    //FB-s
    EL3255_Error    : FB_TerminalError;
    CH1_Error       : FB_GenericError;
    CH2_Error       : FB_GenericError;
    CH3_Error       : FB_GenericError;
    CH4_Error       : FB_GenericError;
    CH5_Error       : FB_GenericError;
END_VAR

(*
* TODO: Test on hardware
*)
EnO:=En;

IF En THEN
    //Channel #1 Status
    IF (wCh1_Status AND 16#2057) <> 0 THEN
        CH1_Error.sErrorMessage := 'EL3255 Channel #1: ';
        IF wCH1_Status.0    THEN    CH1_Error.sErrorMessage := CONCAT(CH1_Error.sErrorMessage, 'Underrange; ');             IF CH1_Error.ErrorPriority > 100 OR CH1_Error.ErrorPriority = 0     THEN CH1_Error.ErrorPriority := 100;    END_IF      END_IF
        IF wCH1_Status.1    THEN    CH1_Error.sErrorMessage := CONCAT(CH1_Error.sErrorMessage, 'Overrange; ');              IF CH1_Error.ErrorPriority > 100 OR CH1_Error.ErrorPriority = 0     THEN CH1_Error.ErrorPriority := 100;    END_IF      END_IF
        IF wCh1_Status.2    THEN    CH1_Error.sErrorMessage := CONCAT(CH1_Error.sErrorMessage, 'Limit 1; ');                IF CH1_Error.ErrorPriority > 100 OR CH1_Error.ErrorPriority = 0     THEN CH1_Error.ErrorPriority := 100;    END_IF      END_IF
        IF wCh1_Status.4    THEN    CH1_Error.sErrorMessage := CONCAT(CH1_Error.sErrorMessage, 'Limit 2; ');                IF CH1_Error.ErrorPriority > 100 OR CH1_Error.ErrorPriority = 0     THEN CH1_Error.ErrorPriority := 100;    END_IF      END_IF
        IF wCh1_Status.6    THEN    CH1_Error.sErrorMessage := CONCAT(CH1_Error.sErrorMessage, 'Error; ');                  IF CH1_Error.ErrorPriority > 10  OR CH1_Error.ErrorPriority = 0     THEN CH1_Error.ErrorPriority := 10;     END_IF      END_IF
        IF wCh1_Status.13   THEN    CH1_Error.sErrorMessage := CONCAT(CH1_Error.sErrorMessage, 'Sync error; ');             IF CH1_Error.ErrorPriority > 10  OR CH1_Error.ErrorPriority = 0     THEN CH1_Error.ErrorPriority := 10;     END_IF      END_IF
        CH1_Error.bError := TRUE;
    ELSE
        CH1_Error.bError        := FALSE;
        CH1_Error.sErrorMessage := '';
    END_IF

    //Channel #2 Status
    IF (wCh2_Status AND 16#2057) <> 0 THEN
        CH2_Error.sErrorMessage := 'EL3255 Channel #2: ';
        IF wCH2_Status.0    THEN    CH2_Error.sErrorMessage := CONCAT(CH2_Error.sErrorMessage, 'Underrange; ');             IF CH2_Error.ErrorPriority > 100 OR CH2_Error.ErrorPriority = 0     THEN CH2_Error.ErrorPriority := 100;    END_IF      END_IF
        IF wCH2_Status.1    THEN    CH2_Error.sErrorMessage := CONCAT(CH2_Error.sErrorMessage, 'Overrange; ');              IF CH2_Error.ErrorPriority > 100 OR CH2_Error.ErrorPriority = 0     THEN CH2_Error.ErrorPriority := 100;    END_IF      END_IF
        IF wCh2_Status.2    THEN    CH2_Error.sErrorMessage := CONCAT(CH2_Error.sErrorMessage, 'Limit 1; ');                IF CH2_Error.ErrorPriority > 100 OR CH2_Error.ErrorPriority = 0     THEN CH2_Error.ErrorPriority := 100;    END_IF      END_IF
        IF wCh2_Status.4    THEN    CH2_Error.sErrorMessage := CONCAT(CH2_Error.sErrorMessage, 'Limit 2; ');                IF CH2_Error.ErrorPriority > 100 OR CH2_Error.ErrorPriority = 0     THEN CH2_Error.ErrorPriority := 100;    END_IF      END_IF
        IF wCh2_Status.6    THEN    CH2_Error.sErrorMessage := CONCAT(CH2_Error.sErrorMessage, 'Error; ');                  IF CH2_Error.ErrorPriority > 10  OR CH2_Error.ErrorPriority = 0     THEN CH2_Error.ErrorPriority := 10;     END_IF      END_IF
        IF wCh2_Status.13   THEN    CH2_Error.sErrorMessage := CONCAT(CH2_Error.sErrorMessage, 'Sync error; ');             IF CH2_Error.ErrorPriority > 10  OR CH2_Error.ErrorPriority = 0     THEN CH2_Error.ErrorPriority := 10;     END_IF      END_IF
        CH2_Error.bError := TRUE;
    ELSE
        CH2_Error.bError        := FALSE;
        CH2_Error.sErrorMessage := '';
    END_IF

    //Channel #3 Status
    IF (wCh3_Status AND 16#2057) <> 0 THEN
        CH3_Error.sErrorMessage := 'EL3255 Channel #3: ';
        IF wCH3_Status.0    THEN    CH3_Error.sErrorMessage := CONCAT(CH3_Error.sErrorMessage, 'Underrange; ');             IF CH3_Error.ErrorPriority > 100 OR CH3_Error.ErrorPriority = 0     THEN CH3_Error.ErrorPriority := 100;    END_IF      END_IF
        IF wCH3_Status.1    THEN    CH3_Error.sErrorMessage := CONCAT(CH3_Error.sErrorMessage, 'Overrange; ');              IF CH3_Error.ErrorPriority > 100 OR CH3_Error.ErrorPriority = 0     THEN CH3_Error.ErrorPriority := 100;    END_IF      END_IF
        IF wCh3_Status.2    THEN    CH3_Error.sErrorMessage := CONCAT(CH3_Error.sErrorMessage, 'Limit 1; ');                IF CH3_Error.ErrorPriority > 100 OR CH3_Error.ErrorPriority = 0     THEN CH3_Error.ErrorPriority := 100;    END_IF      END_IF
        IF wCh3_Status.4    THEN    CH3_Error.sErrorMessage := CONCAT(CH3_Error.sErrorMessage, 'Limit 2; ');                IF CH3_Error.ErrorPriority > 100 OR CH3_Error.ErrorPriority = 0     THEN CH3_Error.ErrorPriority := 100;    END_IF      END_IF
        IF wCh3_Status.6    THEN    CH3_Error.sErrorMessage := CONCAT(CH3_Error.sErrorMessage, 'Error; ');                  IF CH3_Error.ErrorPriority > 10  OR CH3_Error.ErrorPriority = 0     THEN CH3_Error.ErrorPriority := 10;     END_IF      END_IF
        IF wCh3_Status.13   THEN    CH3_Error.sErrorMessage := CONCAT(CH3_Error.sErrorMessage, 'Sync error; ');             IF CH3_Error.ErrorPriority > 10  OR CH3_Error.ErrorPriority = 0     THEN CH3_Error.ErrorPriority := 10;     END_IF      END_IF
        CH3_Error.bError := TRUE;
    ELSE
        CH3_Error.bError        := FALSE;
        CH3_Error.sErrorMessage := '';
    END_IF

    //Channel #4 Status
    IF (wCh4_Status AND 16#2057) <> 0 THEN
        CH4_Error.sErrorMessage := 'EL3255 Channel #4: ';
        IF wCH4_Status.0    THEN    CH4_Error.sErrorMessage := CONCAT(CH4_Error.sErrorMessage, 'Underrange; ');             IF CH4_Error.ErrorPriority > 100 OR CH4_Error.ErrorPriority = 0     THEN CH4_Error.ErrorPriority := 100;    END_IF      END_IF
        IF wCH4_Status.1    THEN    CH4_Error.sErrorMessage := CONCAT(CH4_Error.sErrorMessage, 'Overrange; ');              IF CH4_Error.ErrorPriority > 100 OR CH4_Error.ErrorPriority = 0     THEN CH4_Error.ErrorPriority := 100;    END_IF      END_IF
        IF wCh4_Status.2    THEN    CH4_Error.sErrorMessage := CONCAT(CH4_Error.sErrorMessage, 'Limit 1; ');                IF CH4_Error.ErrorPriority > 100 OR CH4_Error.ErrorPriority = 0     THEN CH4_Error.ErrorPriority := 100;    END_IF      END_IF
        IF wCh4_Status.4    THEN    CH4_Error.sErrorMessage := CONCAT(CH4_Error.sErrorMessage, 'Limit 2; ');                IF CH4_Error.ErrorPriority > 100 OR CH4_Error.ErrorPriority = 0     THEN CH4_Error.ErrorPriority := 100;    END_IF      END_IF
        IF wCh4_Status.6    THEN    CH4_Error.sErrorMessage := CONCAT(CH4_Error.sErrorMessage, 'Error; ');                  IF CH4_Error.ErrorPriority > 10  OR CH4_Error.ErrorPriority = 0     THEN CH4_Error.ErrorPriority := 10;     END_IF      END_IF
        IF wCh4_Status.13   THEN    CH4_Error.sErrorMessage := CONCAT(CH4_Error.sErrorMessage, 'Sync error; ');             IF CH4_Error.ErrorPriority > 10  OR CH4_Error.ErrorPriority = 0     THEN CH4_Error.ErrorPriority := 10;     END_IF      END_IF
        CH4_Error.bError := TRUE;
    ELSE
        CH4_Error.bError        := FALSE;
        CH4_Error.sErrorMessage := '';
    END_IF

    //Channel #5 Status
    IF (wCh5_Status AND 16#2057) <> 0 THEN
        CH5_Error.sErrorMessage := 'EL3255 Channel #5: ';
        IF wCH5_Status.0    THEN    CH5_Error.sErrorMessage := CONCAT(CH5_Error.sErrorMessage, 'Underrange; ');             IF CH5_Error.ErrorPriority > 100 OR CH5_Error.ErrorPriority = 0     THEN CH5_Error.ErrorPriority := 100;    END_IF      END_IF
        IF wCH5_Status.1    THEN    CH5_Error.sErrorMessage := CONCAT(CH5_Error.sErrorMessage, 'Overrange; ');              IF CH5_Error.ErrorPriority > 100 OR CH5_Error.ErrorPriority = 0     THEN CH5_Error.ErrorPriority := 100;    END_IF      END_IF
        IF wCh5_Status.2    THEN    CH5_Error.sErrorMessage := CONCAT(CH5_Error.sErrorMessage, 'Limit 1; ');                IF CH5_Error.ErrorPriority > 100 OR CH5_Error.ErrorPriority = 0     THEN CH5_Error.ErrorPriority := 100;    END_IF      END_IF
        IF wCh5_Status.4    THEN    CH5_Error.sErrorMessage := CONCAT(CH5_Error.sErrorMessage, 'Limit 2; ');                IF CH5_Error.ErrorPriority > 100 OR CH5_Error.ErrorPriority = 0     THEN CH5_Error.ErrorPriority := 100;    END_IF      END_IF
        IF wCh5_Status.6    THEN    CH5_Error.sErrorMessage := CONCAT(CH5_Error.sErrorMessage, 'Error; ');                  IF CH5_Error.ErrorPriority > 10  OR CH5_Error.ErrorPriority = 0     THEN CH5_Error.ErrorPriority := 10;     END_IF      END_IF
        IF wCh5_Status.13   THEN    CH5_Error.sErrorMessage := CONCAT(CH5_Error.sErrorMessage, 'Sync error; ');             IF CH5_Error.ErrorPriority > 10  OR CH5_Error.ErrorPriority = 0     THEN CH5_Error.ErrorPriority := 10;     END_IF      END_IF
        CH5_Error.bError := TRUE;
    ELSE
        CH5_Error.bError        := FALSE;
        CH5_Error.sErrorMessage := '';
    END_IF

END_IF

//Error FB instance
EL3255_Error(
    En                  := TRUE,
    iTerminal_ID        := iTerminal_ID,
    bWcState            := WcState_WcState,
    uiInfoData_State    := InfoData_State,
    pErrorSystem        := ErrorSystem,
    bError              => bError,
);

CH1_Error (
    En              := En,
    bError          := ,
    sErrorMessage   := ,
    ErrorPriority   := ,
    iTerminal_ID    := iTerminal_ID,
    pErrorSystem    := ErrorSystem,
    EnO             => ,
);

CH2_Error (
    En              := En,
    bError          := ,
    sErrorMessage   := ,
    ErrorPriority   := ,
    iTerminal_ID    := iTerminal_ID,
    pErrorSystem    := ErrorSystem,
    EnO             => ,
);

CH3_Error (
    En              := En,
    bError          := ,
    sErrorMessage   := ,
    ErrorPriority   := ,
    iTerminal_ID    := iTerminal_ID,
    pErrorSystem    := ErrorSystem,
    EnO             => ,
);

CH4_Error (
    En              := En,
    bError          := ,
    sErrorMessage   := ,
    ErrorPriority   := ,
    iTerminal_ID    := iTerminal_ID,
    pErrorSystem    := ErrorSystem,
    EnO             => ,
);

CH5_Error (
    En              := En,
    bError          := ,
    sErrorMessage   := ,
    ErrorPriority   := ,
    iTerminal_ID    := iTerminal_ID,
    pErrorSystem    := ErrorSystem,
    EnO             => ,
);

END_FUNCTION_BLOCK

// ---- tc_mca_std_lib/POUs/Hardware/EtherCAT_Terminals/Digital_Inputs/EL1008.TcPOU
///EL1008 | 8-channel digital input terminal 24 V DC, 3 ms
FUNCTION_BLOCK EL1008

VAR_INPUT
    En              : BOOL;
    iTerminal_ID    : INT;
    ErrorSystem     : POINTER TO ST_ErrorSystem;
END_VAR

VAR_OUTPUT
    EnO     : BOOL;
    bError  : BOOL;
END_VAR

VAR
    WcState_WcState     AT %I*  : BOOL;
    InfoData_State      AT %I*  : UINT;

    //FB-s
    EL1008_Error    : FB_TerminalError;
END_VAR

(*
* TODO: DONE!
*)
EnO:=En;

//Error FB instance
EL1008_Error(
    En                  := TRUE,
    iTerminal_ID        := iTerminal_ID,
    bWcState            := WcState_WcState,
    uiInfoData_State    := InfoData_State,
    pErrorSystem        := ErrorSystem,
    bError              => bError,
);

END_FUNCTION_BLOCK

// ---- tc_mca_std_lib/POUs/Hardware/EtherCAT_Terminals/Digital_Inputs/EL1018.TcPOU
///EL1018 | 8-channel digital input terminal 24 V DC, 10 µs
FUNCTION_BLOCK EL1018

VAR_INPUT
    En              : BOOL;
    iTerminal_ID    : INT;
    ErrorSystem     : POINTER TO ST_ErrorSystem;
END_VAR

VAR_OUTPUT
    EnO         : BOOL;
    bError      : BOOL;
END_VAR

VAR
    WcState_WcState     AT %I*  : BOOL;
    InfoData_State      AT %I*  : UINT;

    //FB-s
    EL1018_Error    : FB_TerminalError;
END_VAR

(*
* TODO: DONE!
*)
EnO:=En;

//Error FB instance
EL1018_Error(
    En                  := TRUE,
    iTerminal_ID        := iTerminal_ID,
    bWcState            := WcState_WcState,
    uiInfoData_State    := InfoData_State,
    pErrorSystem        := ErrorSystem,
    bError              => bError,
);

END_FUNCTION_BLOCK

// ---- tc_mca_std_lib/POUs/Hardware/EtherCAT_Terminals/Digital_Inputs/EL1252.TcPOU
//EL1252 or EL1252-0050 | 2-channel digitl input terminal with timestamp
FUNCTION_BLOCK EL1252
VAR_INPUT
    En              : BOOL;
    iTerminal_ID    : INT;
    ErrorSystem     : POINTER TO ST_ErrorSystem;
END_VAR

VAR_OUTPUT
    EnO     : BOOL;
    bError  : BOOL;
END_VAR

VAR
    WcState_WcState     AT %I*  : BOOL;
    InfoData_State      AT %I*  : UINT;

    //FB-s
    EL1252_Error        : FB_TerminalError;
END_VAR

(*
* TODO: DONE!
*)
EnO:=En;

//Error FB instance
EL1252_Error(
    En                  := TRUE,
    iTerminal_ID        := iTerminal_ID,
    bWcState            := WcState_WcState,
    uiInfoData_State    := InfoData_State,
    pErrorSystem        := ErrorSystem,
    bError              => bError,
);

END_FUNCTION_BLOCK

// ---- tc_mca_std_lib/POUs/Hardware/EtherCAT_Terminals/Digital_Inputs/EL1808.TcPOU
///EL1808 | HD EtherCAT Terminals, 8-channel digital input 24 V DC, 3 ms, 2-wire connection
FUNCTION_BLOCK EL1808

VAR_INPUT
    En              : BOOL;
    iTerminal_ID    : INT;
    ErrorSystem     : POINTER TO ST_ErrorSystem;
END_VAR

VAR_OUTPUT
    EnO         : BOOL;
    bError      : BOOL;
END_VAR

VAR
    WcState_WcState     AT %I*  : BOOL;
    InfoData_State      AT %I*  : UINT;

    //FB-s
    EL1808_Error    : FB_TerminalError;
END_VAR

(*
* TODO: DONE!
*)
EnO:=En;

//Error FB instance
EL1808_Error(
    En                  := TRUE,
    iTerminal_ID        := iTerminal_ID,
    bWcState            := WcState_WcState,
    uiInfoData_State    := InfoData_State,
    pErrorSystem        := ErrorSystem,
    bError              => bError,
);

END_FUNCTION_BLOCK

// ---- tc_mca_std_lib/POUs/Hardware/EtherCAT_Terminals/Digital_Inputs/EL1809.TcPOU
///EL1809 | HD EtherCAT Terminals, 16-channel digital input 24 V DC, 3 ms
FUNCTION_BLOCK EL1809

VAR_INPUT
    En              : BOOL;
    iTerminal_ID    : INT;
    ErrorSystem     : POINTER TO ST_ErrorSystem;
END_VAR

VAR_OUTPUT
    EnO     : BOOL;
    bError  : BOOL;
END_VAR

VAR
    WcState_WcState     AT %I*  : BOOL;
    InfoData_State      AT %I*  : UINT;

    //FB-s
    EL1809_Error    : FB_TerminalError;
END_VAR

(*
* TODO: DONE!
*)
EnO:=En;

//Error FB instance
EL1809_Error(
    En                  := TRUE,
    iTerminal_ID        := iTerminal_ID,
    bWcState            := WcState_WcState,
    uiInfoData_State    := InfoData_State,
    pErrorSystem        := ErrorSystem,
    bError              => bError,
);

END_FUNCTION_BLOCK

// ---- tc_mca_std_lib/POUs/Hardware/EtherCAT_Terminals/Digital_Inputs/EL1819.TcPOU
///EL1819 | HD EtherCAT Terminals, 16-channel digital input 24 V DC, 10 µs
FUNCTION_BLOCK EL1819

VAR_INPUT
    En              : BOOL;
    iTerminal_ID    : INT;
    ErrorSystem     : POINTER TO ST_ErrorSystem;
END_VAR

VAR_OUTPUT
    EnO         : BOOL;
    bError      : BOOL;
END_VAR

VAR
    WcState_WcState     AT %I*  : BOOL;
    InfoData_State      AT %I*  : UINT;

    //FB-s
    EL1819_Error    : FB_TerminalError;
END_VAR

(*
* TODO: DONE!
*)
EnO:=En;

//Error FB instance
EL1819_Error(
    En                  := TRUE,
    iTerminal_ID        := iTerminal_ID,
    bWcState            := WcState_WcState,
    uiInfoData_State    := InfoData_State,
    pErrorSystem        := ErrorSystem,
    bError              => bError,
);

END_FUNCTION_BLOCK

// ---- tc_mca_std_lib/POUs/Hardware/EtherCAT_Terminals/Digital_Outputs/EL2014.TcPOU
// EL2014 | 4-channel output terminal, 24V DC, 0.5A, 4 x 0V contact
FUNCTION_BLOCK EL2014
VAR_INPUT
    En              : BOOL;
    iTerminal_ID    : INT;
    ErrorSystem     : POINTER TO ST_ErrorSystem;
END_VAR

VAR_OUTPUT
    EnO         : BOOL;
    bError      : BOOL;
END_VAR

VAR
    //Channel Diagnostic Inputs
    wCH1_Diag       AT %I*  : BYTE;
    wCH2_Diag       AT %I*  : BYTE;
    wCH3_Diag       AT %I*  : BYTE;
    wCH4_Diag       AT %I*  : BYTE;
    //Device Diagnostic Inputs
    wDevice_Diag        AT %I*  : BYTE;
    //Device State Inputs
    WcState_WcState     AT %I*  : BOOL;
    InfoData_State      AT %I*  : UINT;


    //FB-s
    EL2014_Error    : FB_TerminalError;
    CH1_Error       : FB_GenericError;
    CH2_Error       : FB_GenericError;
    CH3_Error       : FB_GenericError;
    CH4_Error       : FB_GenericError;
    DEV_Error       : FB_GenericError;
END_VAR

(*
*   TODO: Test on hardware
*)
EnO:=En;

IF En THEN

    //Channel #1 Diag
    IF wCH1_Diag <> 0 THEN
        CH1_Error.sErrorMessage := 'EL2014 Channel #1: ';
        IF wCH1_Diag.0  THEN    CH1_Error.sErrorMessage := CONCAT(CH1_Error.sErrorMessage, 'Overtemperature; ');            IF CH1_Error.ErrorPriority > 10  OR CH1_Error.ErrorPriority = 0     THEN CH1_Error.ErrorPriority := 10;     END_IF      END_IF
        IF wCH1_Diag.1  THEN    CH1_Error.sErrorMessage := CONCAT(CH1_Error.sErrorMessage, 'Open Load; ');                  IF CH1_Error.ErrorPriority > 100 OR CH1_Error.ErrorPriority = 0     THEN CH1_Error.ErrorPriority := 100;    END_IF      END_IF
        IF wCH1_Diag.2  THEN    CH1_Error.sErrorMessage := CONCAT(CH1_Error.sErrorMessage, 'Overcurrent; ');                IF CH1_Error.ErrorPriority > 10  OR CH1_Error.ErrorPriority = 0     THEN CH1_Error.ErrorPriority := 10;     END_IF      END_IF
        IF wCH1_Diag.3  THEN    CH1_Error.sErrorMessage := CONCAT(CH1_Error.sErrorMessage, 'Short Circuit to 24V; ');       IF CH1_Error.ErrorPriority > 10  OR CH1_Error.ErrorPriority = 0     THEN CH1_Error.ErrorPriority := 10;     END_IF      END_IF
        CH1_Error.bError := TRUE;
    ELSE
        CH1_Error.bError := FALSE;
        CH1_Error.sErrorMessage := '';
    END_IF

    //Channel #2 Diag
    IF wCH2_Diag <> 0 THEN
        CH2_Error.sErrorMessage := 'EL2014 Channel #2: ';
        IF wCH2_Diag.0  THEN    CH2_Error.sErrorMessage := CONCAT(CH2_Error.sErrorMessage, 'Overtemperature; ');            IF CH2_Error.ErrorPriority > 10  OR CH2_Error.ErrorPriority = 0     THEN CH2_Error.ErrorPriority := 10;     END_IF      END_IF
        IF wCH2_Diag.1  THEN    CH2_Error.sErrorMessage := CONCAT(CH2_Error.sErrorMessage, 'Open Load; ');                  IF CH2_Error.ErrorPriority > 100 OR CH2_Error.ErrorPriority = 0     THEN CH2_Error.ErrorPriority := 100;    END_IF      END_IF
        IF wCH2_Diag.2  THEN    CH2_Error.sErrorMessage := CONCAT(CH2_Error.sErrorMessage, 'Overcurrent; ');                IF CH2_Error.ErrorPriority > 10  OR CH2_Error.ErrorPriority = 0     THEN CH2_Error.ErrorPriority := 10;     END_IF      END_IF
        IF wCH2_Diag.3  THEN    CH2_Error.sErrorMessage := CONCAT(CH2_Error.sErrorMessage, 'Short Circuit to 24V; ');       IF CH2_Error.ErrorPriority > 10  OR CH2_Error.ErrorPriority = 0     THEN CH2_Error.ErrorPriority := 10;     END_IF      END_IF
        CH2_Error.bError := TRUE;
    ELSE
        CH2_Error.bError := FALSE;
        CH2_Error.sErrorMessage := '';
    END_IF

    //Channel #3 Diag
    IF wCH3_Diag <> 0 THEN
        CH3_Error.sErrorMessage := 'EL2014 Channel #3: ';
        IF wCH3_Diag.0  THEN    CH3_Error.sErrorMessage := CONCAT(CH3_Error.sErrorMessage, 'Overtemperature; ');            IF CH3_Error.ErrorPriority > 10  OR CH3_Error.ErrorPriority = 0     THEN CH3_Error.ErrorPriority := 10;     END_IF      END_IF
        IF wCH3_Diag.1  THEN    CH3_Error.sErrorMessage := CONCAT(CH3_Error.sErrorMessage, 'Open Load; ');                  IF CH3_Error.ErrorPriority > 100 OR CH3_Error.ErrorPriority = 0     THEN CH3_Error.ErrorPriority := 100;    END_IF      END_IF
        IF wCH3_Diag.2  THEN    CH3_Error.sErrorMessage := CONCAT(CH3_Error.sErrorMessage, 'Overcurrent; ');                IF CH3_Error.ErrorPriority > 10  OR CH3_Error.ErrorPriority = 0     THEN CH3_Error.ErrorPriority := 10;     END_IF      END_IF
        IF wCH3_Diag.3  THEN    CH3_Error.sErrorMessage := CONCAT(CH3_Error.sErrorMessage, 'Short Circuit to 24V; ');       IF CH3_Error.ErrorPriority > 10  OR CH3_Error.ErrorPriority = 0     THEN CH3_Error.ErrorPriority := 10;     END_IF      END_IF
        CH3_Error.bError := TRUE;
    ELSE
        CH3_Error.bError := FALSE;
        CH3_Error.sErrorMessage := '';
    END_IF

    //Channel #4 Diag
    IF wCH4_Diag <> 0 THEN
        CH4_Error.sErrorMessage := 'EL2014 Channel #4: ';
        IF wCH4_Diag.0  THEN    CH4_Error.sErrorMessage := CONCAT(CH4_Error.sErrorMessage, 'Overtemperature; ');            IF CH4_Error.ErrorPriority > 10  OR CH4_Error.ErrorPriority = 0     THEN CH4_Error.ErrorPriority := 10;     END_IF      END_IF
        IF wCH4_Diag.1  THEN    CH4_Error.sErrorMessage := CONCAT(CH4_Error.sErrorMessage, 'Open Load; ');                  IF CH4_Error.ErrorPriority > 100 OR CH4_Error.ErrorPriority = 0     THEN CH4_Error.ErrorPriority := 100;    END_IF      END_IF
        IF wCH4_Diag.2  THEN    CH4_Error.sErrorMessage := CONCAT(CH4_Error.sErrorMessage, 'Overcurrent; ');                IF CH4_Error.ErrorPriority > 10  OR CH4_Error.ErrorPriority = 0     THEN CH4_Error.ErrorPriority := 10;     END_IF      END_IF
        IF wCH4_Diag.3  THEN    CH4_Error.sErrorMessage := CONCAT(CH4_Error.sErrorMessage, 'Short Circuit to 24V; ');       IF CH4_Error.ErrorPriority > 10  OR CH4_Error.ErrorPriority = 0     THEN CH4_Error.ErrorPriority := 10;     END_IF      END_IF
        CH4_Error.bError := TRUE;
    ELSE
        CH4_Error.bError := FALSE;
        CH4_Error.sErrorMessage := '';
    END_IF

    //Device Diag
    IF wDevice_Diag <> 0 THEN
        DEV_Error.sErrorMessage := 'EL2014: ' ;
        IF wDevice_Diag.0   THEN    DEV_Error.sErrorMessage := CONCAT(DEV_Error.sErrorMessage, 'Common Fault; ');                   IF DEV_Error.ErrorPriority > 100 OR DEV_Error.ErrorPriority = 0     THEN DEV_Error.ErrorPriority := 100;    END_IF      END_IF
        IF wDevice_Diag.1   THEN    DEV_Error.sErrorMessage := CONCAT(DEV_Error.sErrorMessage, 'Device Overtemperature; ');         IF DEV_Error.ErrorPriority > 10  OR DEV_Error.ErrorPriority = 0     THEN DEV_Error.ErrorPriority := 10;     END_IF      END_IF
        IF wDevice_Diag.2   THEN    DEV_Error.sErrorMessage := CONCAT(DEV_Error.sErrorMessage, 'Undervoltage; ');                   IF DEV_Error.ErrorPriority > 10  OR DEV_Error.ErrorPriority = 0     THEN DEV_Error.ErrorPriority := 10;     END_IF      END_IF
        IF wDevice_Diag.3   THEN    DEV_Error.sErrorMessage := CONCAT(DEV_Error.sErrorMessage, 'Missing Voltage; ');                IF DEV_Error.ErrorPriority > 10  OR DEV_Error.ErrorPriority = 0     THEN DEV_Error.ErrorPriority := 10;     END_IF      END_IF
        DEV_Error.bError := TRUE;
    ELSE
        DEV_Error.bError := FALSE;
        DEV_Error.sErrorMessage := '';
    END_IF

END_IF

//Terminal's State of Operation
EL2014_Error(
    En                  := TRUE,
    iTerminal_ID        := iTerminal_ID,
    bWcState            := WcState_WcState,
    uiInfoData_State    := InfoData_State,
    pErrorSystem        := ErrorSystem,
    bError              => bError,
);

CH1_Error (
    En                  :=  En,
    bError              :=  ,
    sErrorMessage       :=  ,
    ErrorPriority       :=  ,
    iTerminal_ID        :=  iTerminal_ID,
    pErrorSystem        :=  ErrorSystem,
    EnO                 =>  ,
);

CH2_Error (
    En                  :=  En,
    bError              :=  ,
    sErrorMessage       :=  ,
    ErrorPriority       :=  ,
    iTerminal_ID        :=  iTerminal_ID,
    pErrorSystem        :=  ErrorSystem,
    EnO                 =>  ,
);

CH3_Error (
    En                  :=  En,
    bError              :=  ,
    sErrorMessage       :=  ,
    ErrorPriority       :=  ,
    iTerminal_ID        :=  iTerminal_ID,
    pErrorSystem        :=  ErrorSystem,
    EnO                 =>  ,
);

CH4_Error (
    En                  :=  En,
    bError              :=  ,
    sErrorMessage       :=  ,
    ErrorPriority       :=  ,
    iTerminal_ID        :=  iTerminal_ID,
    pErrorSystem        :=  ErrorSystem,
    EnO                 =>  ,
);

DEV_Error (
    En                  :=  En,
    bError              :=  ,
    sErrorMessage       :=  ,
    ErrorPriority       :=  ,
    iTerminal_ID        :=  iTerminal_ID,
    pErrorSystem        :=  ErrorSystem,
    EnO                 =>  ,
);

END_FUNCTION_BLOCK

// ---- tc_mca_std_lib/POUs/Hardware/EtherCAT_Terminals/Digital_Outputs/EL2252.TcPOU
///EL2252 | XFC, 2-channel digital output terminal with time stamp, tri-state
FUNCTION_BLOCK EL2252
VAR_INPUT
    En              : BOOL;
    iTerminal_ID    : INT;
    ErrorSystem     : POINTER TO ST_ErrorSystem;
END_VAR

VAR_OUTPUT
    EnO     : BOOL;
    bError  : BOOL;
END_VAR

VAR
    WcState_WcState     AT %I*: BOOL;
    InfoData_State      AT %I*: UINT;

    //FB-s
    EL2252_Error    : FB_TerminalError;
END_VAR

(*
* TODO: DONE!
*)

EL2252_Error(
    En                  := TRUE,
    iTerminal_ID        := iTerminal_ID,
    bWcState            := WcState_WcState,
    uiInfoData_State    := InfoData_State,
    pErrorSystem        := ErrorSystem,
    bError              => bError,
);

END_FUNCTION_BLOCK

// ---- tc_mca_std_lib/POUs/Hardware/EtherCAT_Terminals/Digital_Outputs/EL2808.TcPOU
FUNCTION_BLOCK EL2808

VAR_INPUT
    En              : BOOL;
    iTerminal_ID    : INT;
    ErrorSystem     : POINTER TO ST_ErrorSystem;
END_VAR

VAR_OUTPUT
    EnO     : BOOL;
    bError  : BOOL;
END_VAR

VAR
    WcState_WcState     AT %I*  : BOOL;
    InfoData_State      AT %I*  : UINT;

    //FB-s
    EL2808_Error    : FB_TerminalError;
END_VAR

(*
* TODO: DONE!
*)
EnO:=En;

EL2808_Error(
    En                  := TRUE,
    iTerminal_ID        := iTerminal_ID,
    bWcState            := WcState_WcState,
    uiInfoData_State    := InfoData_State,
    pErrorSystem        := ErrorSystem,
    bError              => bError,
);

END_FUNCTION_BLOCK

// ---- tc_mca_std_lib/POUs/Hardware/EtherCAT_Terminals/Digital_Outputs/EL2819.TcPOU
FUNCTION_BLOCK EL2819
VAR_INPUT
    En              : BOOL;
    iTerminal_ID    : INT;
    ErrorSystem     : POINTER TO ST_ErrorSystem;
END_VAR

VAR_OUTPUT
    EnO     : BOOL;
    bError  : BOOL;
END_VAR

VAR
    wCH1_Diag       AT %I*  : BYTE;
    wCH2_Diag       AT %I*  : BYTE;
    wCH3_Diag       AT %I*  : BYTE;
    wCH4_Diag       AT %I*  : BYTE;
    wCH5_Diag       AT %I*  : BYTE;
    wCH6_Diag       AT %I*  : BYTE;
    wCH7_Diag       AT %I*  : BYTE;
    wCH8_Diag       AT %I*  : BYTE;
    wCH9_Diag       AT %I*  : BYTE;
    wCH10_Diag      AT %I*  : BYTE;
    wCH11_Diag      AT %I*  : BYTE;
    wCH12_Diag      AT %I*  : BYTE;
    wCH13_Diag      AT %I*  : BYTE;
    wCH14_Diag      AT %I*  : BYTE;
    wCH15_Diag      AT %I*  : BYTE;
    wCH16_Diag      AT %I*  : BYTE;

    bDev_CommonFault            AT %I*  : BOOL;
    bDev_Overtemperature        AT %I*  : BOOL;
    bDev_UnderVoltage           AT %I*  : BOOL;
    bDev_MissingVoltage         AT %I*  : BOOL;

    WcState_WcState     AT %I*  : BOOL;
    InfoData_State      AT %I*  : UINT;

    //FB-s
    EL2819_Error    : FB_TerminalError;

    CH1_Error       : FB_GenericError;
    CH2_Error       : FB_GenericError;
    CH3_Error       : FB_GenericError;
    CH4_Error       : FB_GenericError;
    CH5_Error       : FB_GenericError;
    CH6_Error       : FB_GenericError;
    CH7_Error       : FB_GenericError;
    CH8_Error       : FB_GenericError;
    CH9_Error       : FB_GenericError;
    CH10_Error      : FB_GenericError;
    CH11_Error      : FB_GenericError;
    CH12_Error      : FB_GenericError;
    CH13_Error      : FB_GenericError;
    CH14_Error      : FB_GenericError;
    CH15_Error      : FB_GenericError;
    CH16_Error      : FB_GenericError;

    DEV_Error       : FB_GenericError;
END_VAR

(*
* TODO: test on hardware
*)

EnO:=En;

IF En THEN
    //Channel #1 Diag
    IF (wCH1_Diag AND 16#07) <> 0 THEN
        CH1_Error.sErrorMessage := 'EL2819 Channel #1: ';
        IF wCH1_Diag.0  THEN    CH1_Error.sErrorMessage := CONCAT(CH1_Error.sErrorMessage, 'Overtemperature; ');            IF CH1_Error.ErrorPriority > 10  OR CH1_Error.ErrorPriority = 0     THEN CH1_Error.ErrorPriority := 10;     END_IF      END_IF
        IF wCH1_Diag.1  THEN    CH1_Error.sErrorMessage := CONCAT(CH1_Error.sErrorMessage, 'Open Load; ');                  IF CH1_Error.ErrorPriority > 100 OR CH1_Error.ErrorPriority = 0     THEN CH1_Error.ErrorPriority := 100;    END_IF      END_IF
        IF wCH1_Diag.2  THEN    CH1_Error.sErrorMessage := CONCAT(CH1_Error.sErrorMessage, 'Overcurrent; ');                IF CH1_Error.ErrorPriority > 10  OR CH1_Error.ErrorPriority = 0     THEN CH1_Error.ErrorPriority := 10;     END_IF      END_IF
        IF wCH1_Diag.3  THEN    CH1_Error.sErrorMessage := CONCAT(CH1_Error.sErrorMessage, 'Short Circuit to 24V; ');       IF CH1_Error.ErrorPriority > 10  OR CH1_Error.ErrorPriority = 0     THEN CH1_Error.ErrorPriority := 10;     END_IF      END_IF
        CH1_Error.bError := TRUE;
    ELSE
        CH1_Error.bError := FALSE;
        CH1_Error.sErrorMessage := '';
    END_IF

    //Channel #2 Diag
    IF (wCH2_Diag AND 16#07) <> 0 THEN
        CH2_Error.sErrorMessage := 'EL2819 Channel #2: ';
        IF wCH2_Diag.0  THEN    CH2_Error.sErrorMessage := CONCAT(CH2_Error.sErrorMessage, 'Overtemperature; ');            IF CH2_Error.ErrorPriority > 10  OR CH2_Error.ErrorPriority = 0     THEN CH2_Error.ErrorPriority := 10;     END_IF      END_IF
        IF wCH2_Diag.1  THEN    CH2_Error.sErrorMessage := CONCAT(CH2_Error.sErrorMessage, 'Open Load; ');                  IF CH2_Error.ErrorPriority > 100 OR CH2_Error.ErrorPriority = 0     THEN CH2_Error.ErrorPriority := 100;    END_IF      END_IF
        IF wCH2_Diag.2  THEN    CH2_Error.sErrorMessage := CONCAT(CH2_Error.sErrorMessage, 'Overcurrent; ');                IF CH2_Error.ErrorPriority > 10  OR CH2_Error.ErrorPriority = 0     THEN CH2_Error.ErrorPriority := 10;     END_IF      END_IF
        IF wCH2_Diag.3  THEN    CH2_Error.sErrorMessage := CONCAT(CH2_Error.sErrorMessage, 'Short Circuit to 24V; ');       IF CH2_Error.ErrorPriority > 10  OR CH2_Error.ErrorPriority = 0     THEN CH2_Error.ErrorPriority := 10;     END_IF      END_IF
        CH2_Error.bError := TRUE;
    ELSE
        CH2_Error.bError := FALSE;
        CH2_Error.sErrorMessage := '';
    END_IF

    //Channel #3 Diag
    IF wCH3_Diag <> 0 THEN
        CH3_Error.sErrorMessage := 'EL2819 Channel #3: ';
        IF wCH3_Diag.0  THEN    CH3_Error.sErrorMessage := CONCAT(CH3_Error.sErrorMessage, 'Overtemperature; ');            IF CH3_Error.ErrorPriority > 10  OR CH3_Error.ErrorPriority = 0     THEN CH3_Error.ErrorPriority := 10;     END_IF      END_IF
        IF wCH3_Diag.1  THEN    CH3_Error.sErrorMessage := CONCAT(CH3_Error.sErrorMessage, 'Open Load; ');                  IF CH3_Error.ErrorPriority > 100 OR CH3_Error.ErrorPriority = 0     THEN CH3_Error.ErrorPriority := 100;    END_IF      END_IF
        IF wCH3_Diag.2  THEN    CH3_Error.sErrorMessage := CONCAT(CH3_Error.sErrorMessage, 'Overcurrent; ');                IF CH3_Error.ErrorPriority > 10  OR CH3_Error.ErrorPriority = 0     THEN CH3_Error.ErrorPriority := 10;     END_IF      END_IF
        IF wCH3_Diag.3  THEN    CH3_Error.sErrorMessage := CONCAT(CH3_Error.sErrorMessage, 'Short Circuit to 24V; ');       IF CH3_Error.ErrorPriority > 10  OR CH3_Error.ErrorPriority = 0     THEN CH3_Error.ErrorPriority := 10;     END_IF      END_IF
        CH3_Error.bError := TRUE;
    ELSE
        CH3_Error.bError := FALSE;
        CH3_Error.sErrorMessage := '';
    END_IF

    //Channel #4 Diag
    IF wCH4_Diag <> 0 THEN
        CH4_Error.sErrorMessage := 'EL2819 Channel #4: ';
        IF wCH4_Diag.0  THEN    CH4_Error.sErrorMessage := CONCAT(CH4_Error.sErrorMessage, 'Overtemperature; ');            IF CH4_Error.ErrorPriority > 10  OR CH4_Error.ErrorPriority = 0     THEN CH4_Error.ErrorPriority := 10;     END_IF      END_IF
        IF wCH4_Diag.1  THEN    CH4_Error.sErrorMessage := CONCAT(CH4_Error.sErrorMessage, 'Open Load; ');                  IF CH4_Error.ErrorPriority > 100 OR CH4_Error.ErrorPriority = 0     THEN CH4_Error.ErrorPriority := 100;    END_IF      END_IF
        IF wCH4_Diag.2  THEN    CH4_Error.sErrorMessage := CONCAT(CH4_Error.sErrorMessage, 'Overcurrent; ');                IF CH4_Error.ErrorPriority > 10  OR CH4_Error.ErrorPriority = 0     THEN CH4_Error.ErrorPriority := 10;     END_IF      END_IF
        IF wCH4_Diag.3  THEN    CH4_Error.sErrorMessage := CONCAT(CH4_Error.sErrorMessage, 'Short Circuit to 24V; ');       IF CH4_Error.ErrorPriority > 10  OR CH4_Error.ErrorPriority = 0     THEN CH4_Error.ErrorPriority := 10;     END_IF      END_IF
        CH4_Error.bError := TRUE;
    ELSE
        CH4_Error.bError := FALSE;
        CH4_Error.sErrorMessage := '';
    END_IF

    //Channel #5 Diag
    IF wCH5_Diag <> 0 THEN
        CH5_Error.sErrorMessage := 'EL2819 Channel #5: ';
        IF wCH5_Diag.0  THEN    CH5_Error.sErrorMessage := CONCAT(CH5_Error.sErrorMessage, 'Overtemperature; ');            IF CH5_Error.ErrorPriority > 10  OR CH5_Error.ErrorPriority = 0     THEN CH5_Error.ErrorPriority := 10;     END_IF      END_IF
        IF wCH5_Diag.1  THEN    CH5_Error.sErrorMessage := CONCAT(CH5_Error.sErrorMessage, 'Open Load; ');                  IF CH5_Error.ErrorPriority > 100 OR CH5_Error.ErrorPriority = 0     THEN CH5_Error.ErrorPriority := 100;    END_IF      END_IF
        IF wCH5_Diag.2  THEN    CH5_Error.sErrorMessage := CONCAT(CH5_Error.sErrorMessage, 'Overcurrent; ');                IF CH5_Error.ErrorPriority > 10  OR CH5_Error.ErrorPriority = 0     THEN CH5_Error.ErrorPriority := 10;     END_IF      END_IF
        IF wCH5_Diag.3  THEN    CH5_Error.sErrorMessage := CONCAT(CH5_Error.sErrorMessage, 'Short Circuit to 24V; ');       IF CH5_Error.ErrorPriority > 10  OR CH5_Error.ErrorPriority = 0     THEN CH5_Error.ErrorPriority := 10;     END_IF      END_IF
        CH5_Error.bError := TRUE;
    ELSE
        CH5_Error.bError := FALSE;
        CH5_Error.sErrorMessage := '';
    END_IF

    //Channel #6 Diag
    IF wCH6_Diag <> 0 THEN
        CH6_Error.sErrorMessage := 'EL2819 Channel #6: ';
        IF wCH6_Diag.0  THEN    CH6_Error.sErrorMessage := CONCAT(CH6_Error.sErrorMessage, 'Overtemperature; ');            IF CH6_Error.ErrorPriority > 10  OR CH6_Error.ErrorPriority = 0     THEN CH6_Error.ErrorPriority := 10;     END_IF      END_IF
        IF wCH6_Diag.1  THEN    CH6_Error.sErrorMessage := CONCAT(CH6_Error.sErrorMessage, 'Open Load; ');                  IF CH6_Error.ErrorPriority > 100 OR CH6_Error.ErrorPriority = 0     THEN CH6_Error.ErrorPriority := 100;    END_IF      END_IF
        IF wCH6_Diag.2  THEN    CH6_Error.sErrorMessage := CONCAT(CH6_Error.sErrorMessage, 'Overcurrent; ');                IF CH6_Error.ErrorPriority > 10  OR CH6_Error.ErrorPriority = 0     THEN CH6_Error.ErrorPriority := 10;     END_IF      END_IF
        IF wCH6_Diag.3  THEN    CH6_Error.sErrorMessage := CONCAT(CH6_Error.sErrorMessage, 'Short Circuit to 24V; ');       IF CH6_Error.ErrorPriority > 10  OR CH6_Error.ErrorPriority = 0     THEN CH6_Error.ErrorPriority := 10;     END_IF      END_IF
        CH6_Error.bError := TRUE;
    ELSE
        CH6_Error.bError := FALSE;
        CH6_Error.sErrorMessage := '';
    END_IF

    //Channel #7 Diag
    IF wCH7_Diag <> 0 THEN
        CH7_Error.sErrorMessage := 'EL2819 Channel #7: ';
        IF wCH7_Diag.0  THEN    CH7_Error.sErrorMessage := CONCAT(CH7_Error.sErrorMessage, 'Overtemperature; ');            IF CH7_Error.ErrorPriority > 10  OR CH7_Error.ErrorPriority = 0     THEN CH7_Error.ErrorPriority := 10;     END_IF      END_IF
        IF wCH7_Diag.1  THEN    CH7_Error.sErrorMessage := CONCAT(CH7_Error.sErrorMessage, 'Open Load; ');                  IF CH7_Error.ErrorPriority > 100 OR CH7_Error.ErrorPriority = 0     THEN CH7_Error.ErrorPriority := 100;    END_IF      END_IF
        IF wCH7_Diag.2  THEN    CH7_Error.sErrorMessage := CONCAT(CH7_Error.sErrorMessage, 'Overcurrent; ');                IF CH7_Error.ErrorPriority > 10  OR CH7_Error.ErrorPriority = 0     THEN CH7_Error.ErrorPriority := 10;     END_IF      END_IF
        IF wCH7_Diag.3  THEN    CH7_Error.sErrorMessage := CONCAT(CH7_Error.sErrorMessage, 'Short Circuit to 24V; ');       IF CH7_Error.ErrorPriority > 10  OR CH7_Error.ErrorPriority = 0     THEN CH7_Error.ErrorPriority := 10;     END_IF      END_IF
        CH7_Error.bError := TRUE;
    ELSE
        CH7_Error.bError := FALSE;
        CH7_Error.sErrorMessage := '';
    END_IF

    //Channel #8 Diag
    IF wCH8_Diag <> 0 THEN
        CH8_Error.sErrorMessage := 'EL2819 Channel #8: ';
        IF wCH8_Diag.0  THEN    CH8_Error.sErrorMessage := CONCAT(CH8_Error.sErrorMessage, 'Overtemperature; ');            IF CH8_Error.ErrorPriority > 10  OR CH8_Error.ErrorPriority = 0     THEN CH8_Error.ErrorPriority := 10;     END_IF      END_IF
        IF wCH8_Diag.1  THEN    CH8_Error.sErrorMessage := CONCAT(CH8_Error.sErrorMessage, 'Open Load; ');                  IF CH8_Error.ErrorPriority > 100 OR CH8_Error.ErrorPriority = 0     THEN CH8_Error.ErrorPriority := 100;    END_IF      END_IF
        IF wCH8_Diag.2  THEN    CH8_Error.sErrorMessage := CONCAT(CH8_Error.sErrorMessage, 'Overcurrent; ');                IF CH8_Error.ErrorPriority > 10  OR CH8_Error.ErrorPriority = 0     THEN CH8_Error.ErrorPriority := 10;     END_IF      END_IF
        IF wCH8_Diag.3  THEN    CH8_Error.sErrorMessage := CONCAT(CH8_Error.sErrorMessage, 'Short Circuit to 24V; ');       IF CH8_Error.ErrorPriority > 10  OR CH8_Error.ErrorPriority = 0     THEN CH8_Error.ErrorPriority := 10;     END_IF      END_IF
        CH8_Error.bError := TRUE;
    ELSE
        CH8_Error.bError := FALSE;
        CH8_Error.sErrorMessage := '';
    END_IF

    //Channel #9 Diag
    IF wCH9_Diag <> 0 THEN
        CH9_Error.sErrorMessage := 'EL2819 Channel #9: ';
        IF wCH9_Diag.0  THEN    CH9_Error.sErrorMessage := CONCAT(CH9_Error.sErrorMessage, 'Overtemperature; ');            IF CH9_Error.ErrorPriority > 10  OR CH9_Error.ErrorPriority = 0     THEN CH9_Error.ErrorPriority := 10;     END_IF      END_IF
        IF wCH9_Diag.1  THEN    CH9_Error.sErrorMessage := CONCAT(CH9_Error.sErrorMessage, 'Open Load; ');                  IF CH9_Error.ErrorPriority > 100 OR CH9_Error.ErrorPriority = 0     THEN CH9_Error.ErrorPriority := 100;    END_IF      END_IF
        IF wCH9_Diag.2  THEN    CH9_Error.sErrorMessage := CONCAT(CH9_Error.sErrorMessage, 'Overcurrent; ');                IF CH9_Error.ErrorPriority > 10  OR CH9_Error.ErrorPriority = 0     THEN CH9_Error.ErrorPriority := 10;     END_IF      END_IF
        IF wCH9_Diag.3  THEN    CH9_Error.sErrorMessage := CONCAT(CH9_Error.sErrorMessage, 'Short Circuit to 24V; ');       IF CH9_Error.ErrorPriority > 10  OR CH9_Error.ErrorPriority = 0     THEN CH9_Error.ErrorPriority := 10;     END_IF      END_IF
        CH9_Error.bError := TRUE;
    ELSE
        CH9_Error.bError := FALSE;
        CH9_Error.sErrorMessage := '';
    END_IF

    //Channel #10 Diag
    IF wCH10_Diag <> 0 THEN
        CH10_Error.sErrorMessage := 'EL2819 Channel #10: ';
        IF wCH10_Diag.0     THEN    CH10_Error.sErrorMessage := CONCAT(CH10_Error.sErrorMessage, 'Overtemperature; ');          IF CH10_Error.ErrorPriority > 10  OR CH10_Error.ErrorPriority = 0   THEN CH10_Error.ErrorPriority := 10;    END_IF      END_IF
        IF wCH10_Diag.1     THEN    CH10_Error.sErrorMessage := CONCAT(CH10_Error.sErrorMessage, 'Open Load; ');                IF CH10_Error.ErrorPriority > 100 OR CH10_Error.ErrorPriority = 0   THEN CH10_Error.ErrorPriority := 100;   END_IF      END_IF
        IF wCH10_Diag.2     THEN    CH10_Error.sErrorMessage := CONCAT(CH10_Error.sErrorMessage, 'Overcurrent; ');              IF CH10_Error.ErrorPriority > 10  OR CH10_Error.ErrorPriority = 0   THEN CH10_Error.ErrorPriority := 10;    END_IF      END_IF
        IF wCH10_Diag.3     THEN    CH10_Error.sErrorMessage := CONCAT(CH10_Error.sErrorMessage, 'Short Circuit to 24V; ');     IF CH10_Error.ErrorPriority > 10  OR CH10_Error.ErrorPriority = 0   THEN CH10_Error.ErrorPriority := 10;    END_IF      END_IF
        CH10_Error.bError := TRUE;
    ELSE
        CH10_Error.bError := FALSE;
        CH10_Error.sErrorMessage := '';
    END_IF

    //Channel #11 Diag
    IF wCH11_Diag <> 0 THEN
        CH11_Error.sErrorMessage := 'EL2819 Channel #11: ';
        IF wCH11_Diag.0     THEN    CH11_Error.sErrorMessage := CONCAT(CH11_Error.sErrorMessage, 'Overtemperature; ');          IF CH11_Error.ErrorPriority > 10  OR CH11_Error.ErrorPriority = 0   THEN CH11_Error.ErrorPriority := 10;    END_IF      END_IF
        IF wCH11_Diag.1     THEN    CH11_Error.sErrorMessage := CONCAT(CH11_Error.sErrorMessage, 'Open Load; ');                IF CH11_Error.ErrorPriority > 100 OR CH11_Error.ErrorPriority = 0   THEN CH11_Error.ErrorPriority := 100;   END_IF      END_IF
        IF wCH11_Diag.2     THEN    CH11_Error.sErrorMessage := CONCAT(CH11_Error.sErrorMessage, 'Overcurrent; ');              IF CH11_Error.ErrorPriority > 10  OR CH11_Error.ErrorPriority = 0   THEN CH11_Error.ErrorPriority := 10;    END_IF      END_IF
        IF wCH11_Diag.3     THEN    CH11_Error.sErrorMessage := CONCAT(CH11_Error.sErrorMessage, 'Short Circuit to 24V; ');     IF CH11_Error.ErrorPriority > 10  OR CH11_Error.ErrorPriority = 0   THEN CH11_Error.ErrorPriority := 10;    END_IF      END_IF
        CH11_Error.bError := TRUE;
    ELSE
        CH11_Error.bError := FALSE;
        CH11_Error.sErrorMessage := '';
    END_IF

    //Channel #12 Diag
    IF wCH12_Diag <> 0 THEN
        CH12_Error.sErrorMessage := 'EL2819 Channel #12: ';
        IF wCH12_Diag.0     THEN    CH12_Error.sErrorMessage := CONCAT(CH12_Error.sErrorMessage, 'Overtemperature; ');          IF CH12_Error.ErrorPriority > 10  OR CH12_Error.ErrorPriority = 0   THEN CH12_Error.ErrorPriority := 10;    END_IF      END_IF
        IF wCH12_Diag.1     THEN    CH12_Error.sErrorMessage := CONCAT(CH12_Error.sErrorMessage, 'Open Load; ');                IF CH12_Error.ErrorPriority > 100 OR CH12_Error.ErrorPriority = 0   THEN CH12_Error.ErrorPriority := 100;   END_IF      END_IF
        IF wCH12_Diag.2     THEN    CH12_Error.sErrorMessage := CONCAT(CH12_Error.sErrorMessage, 'Overcurrent; ');              IF CH12_Error.ErrorPriority > 10  OR CH12_Error.ErrorPriority = 0   THEN CH12_Error.ErrorPriority := 10;    END_IF      END_IF
        IF wCH12_Diag.3     THEN    CH12_Error.sErrorMessage := CONCAT(CH12_Error.sErrorMessage, 'Short Circuit to 24V; ');     IF CH12_Error.ErrorPriority > 10  OR CH12_Error.ErrorPriority = 0   THEN CH12_Error.ErrorPriority := 10;    END_IF      END_IF
        CH12_Error.bError := TRUE;
    ELSE
        CH12_Error.bError := FALSE;
        CH12_Error.sErrorMessage := '';
    END_IF

    //Channel #13 Diag
    IF wCH13_Diag <> 0 THEN
        CH13_Error.sErrorMessage := 'EL2819 Channel #13: ';
        IF wCH13_Diag.0     THEN    CH13_Error.sErrorMessage := CONCAT(CH13_Error.sErrorMessage, 'Overtemperature; ');          IF CH13_Error.ErrorPriority > 10  OR CH13_Error.ErrorPriority = 0   THEN CH13_Error.ErrorPriority := 10;    END_IF      END_IF
        IF wCH13_Diag.1     THEN    CH13_Error.sErrorMessage := CONCAT(CH13_Error.sErrorMessage, 'Open Load; ');                IF CH13_Error.ErrorPriority > 100 OR CH13_Error.ErrorPriority = 0   THEN CH13_Error.ErrorPriority := 100;   END_IF      END_IF
        IF wCH13_Diag.2     THEN    CH13_Error.sErrorMessage := CONCAT(CH13_Error.sErrorMessage, 'Overcurrent; ');              IF CH13_Error.ErrorPriority > 10  OR CH13_Error.ErrorPriority = 0   THEN CH13_Error.ErrorPriority := 10;    END_IF      END_IF
        IF wCH13_Diag.3     THEN    CH13_Error.sErrorMessage := CONCAT(CH13_Error.sErrorMessage, 'Short Circuit to 24V; ');     IF CH13_Error.ErrorPriority > 10  OR CH13_Error.ErrorPriority = 0   THEN CH13_Error.ErrorPriority := 10;    END_IF      END_IF
        CH13_Error.bError := TRUE;
    ELSE
        CH13_Error.bError := FALSE;
        CH13_Error.sErrorMessage := '';
    END_IF

    //Channel #14 Diag
    IF wCH14_Diag <> 0 THEN
        CH14_Error.sErrorMessage := 'EL2819 Channel #14: ';
        IF wCH14_Diag.0     THEN    CH14_Error.sErrorMessage := CONCAT(CH14_Error.sErrorMessage, 'Overtemperature; ');          IF CH14_Error.ErrorPriority > 10  OR CH14_Error.ErrorPriority = 0   THEN CH14_Error.ErrorPriority := 10;    END_IF      END_IF
        IF wCH14_Diag.1     THEN    CH14_Error.sErrorMessage := CONCAT(CH14_Error.sErrorMessage, 'Open Load; ');                IF CH14_Error.ErrorPriority > 100 OR CH14_Error.ErrorPriority = 0   THEN CH14_Error.ErrorPriority := 100;   END_IF      END_IF
        IF wCH14_Diag.2     THEN    CH14_Error.sErrorMessage := CONCAT(CH14_Error.sErrorMessage, 'Overcurrent; ');              IF CH14_Error.ErrorPriority > 10  OR CH14_Error.ErrorPriority = 0   THEN CH14_Error.ErrorPriority := 10;    END_IF      END_IF
        IF wCH14_Diag.3     THEN    CH14_Error.sErrorMessage := CONCAT(CH14_Error.sErrorMessage, 'Short Circuit to 24V; ');     IF CH14_Error.ErrorPriority > 10  OR CH14_Error.ErrorPriority = 0   THEN CH14_Error.ErrorPriority := 10;    END_IF      END_IF
        CH14_Error.bError := TRUE;
    ELSE
        CH14_Error.bError := FALSE;
        CH14_Error.sErrorMessage := '';
    END_IF

    //Channel #15 Diag
    IF wCH15_Diag <> 0 THEN
        CH15_Error.sErrorMessage := 'EL2819 Channel #15: ';
        IF wCH15_Diag.0     THEN    CH15_Error.sErrorMessage := CONCAT(CH15_Error.sErrorMessage, 'Overtemperature; ');          IF CH15_Error.ErrorPriority > 10  OR CH15_Error.ErrorPriority = 0   THEN CH15_Error.ErrorPriority := 10;    END_IF      END_IF
        IF wCH15_Diag.1     THEN    CH15_Error.sErrorMessage := CONCAT(CH15_Error.sErrorMessage, 'Open Load; ');                IF CH15_Error.ErrorPriority > 100 OR CH15_Error.ErrorPriority = 0   THEN CH15_Error.ErrorPriority := 100;   END_IF      END_IF
        IF wCH15_Diag.2     THEN    CH15_Error.sErrorMessage := CONCAT(CH15_Error.sErrorMessage, 'Overcurrent; ');              IF CH15_Error.ErrorPriority > 10  OR CH15_Error.ErrorPriority = 0   THEN CH15_Error.ErrorPriority := 10;    END_IF      END_IF
        IF wCH15_Diag.3     THEN    CH15_Error.sErrorMessage := CONCAT(CH15_Error.sErrorMessage, 'Short Circuit to 24V; ');     IF CH15_Error.ErrorPriority > 10  OR CH15_Error.ErrorPriority = 0   THEN CH15_Error.ErrorPriority := 10;    END_IF      END_IF
        CH15_Error.bError := TRUE;
    ELSE
        CH15_Error.bError := FALSE;
        CH15_Error.sErrorMessage := '';
    END_IF

    //Channel #16 Diag
    IF wCH16_Diag <> 0 THEN
        CH16_Error.sErrorMessage := 'EL2819 Channel #16: ';
        IF wCH16_Diag.0     THEN    CH16_Error.sErrorMessage := CONCAT(CH16_Error.sErrorMessage, 'Overtemperature; ');          IF CH16_Error.ErrorPriority > 10  OR CH16_Error.ErrorPriority = 0   THEN CH16_Error.ErrorPriority := 10;    END_IF      END_IF
        IF wCH16_Diag.1     THEN    CH16_Error.sErrorMessage := CONCAT(CH16_Error.sErrorMessage, 'Open Load; ');                IF CH16_Error.ErrorPriority > 100 OR CH16_Error.ErrorPriority = 0   THEN CH16_Error.ErrorPriority := 100;   END_IF      END_IF
        IF wCH16_Diag.2     THEN    CH16_Error.sErrorMessage := CONCAT(CH16_Error.sErrorMessage, 'Overcurrent; ');              IF CH16_Error.ErrorPriority > 10  OR CH16_Error.ErrorPriority = 0   THEN CH16_Error.ErrorPriority := 10;    END_IF      END_IF
        IF wCH16_Diag.3     THEN    CH16_Error.sErrorMessage := CONCAT(CH16_Error.sErrorMessage, 'Short Circuit to 24V; ');     IF CH16_Error.ErrorPriority > 10  OR CH16_Error.ErrorPriority = 0   THEN CH16_Error.ErrorPriority := 10;    END_IF      END_IF
        CH16_Error.bError := TRUE;
    ELSE
        CH16_Error.bError := FALSE;
        CH16_Error.sErrorMessage := '';
    END_IF

    //Device Diag
    IF bDev_CommonFault OR bDev_Overtemperature OR bDev_UnderVoltage OR bDev_MissingVoltage THEN
        DEV_Error.sErrorMessage := 'EL2819: ' ;
        IF bDev_CommonFault         THEN    DEV_Error.sErrorMessage := CONCAT(DEV_Error.sErrorMessage, 'Common Fault; ');               IF DEV_Error.ErrorPriority > 50  OR DEV_Error.ErrorPriority = 0 THEN DEV_Error.ErrorPriority := 50; END_IF      END_IF
        IF bDev_Overtemperature     THEN    DEV_Error.sErrorMessage := CONCAT(DEV_Error.sErrorMessage, 'Device Overtemperature; ');     IF DEV_Error.ErrorPriority > 10  OR DEV_Error.ErrorPriority = 0 THEN DEV_Error.ErrorPriority := 10; END_IF      END_IF
        IF bDev_UnderVoltage        THEN    DEV_Error.sErrorMessage := CONCAT(DEV_Error.sErrorMessage, 'Undervoltage; ');               IF DEV_Error.ErrorPriority > 10  OR DEV_Error.ErrorPriority = 0 THEN DEV_Error.ErrorPriority := 10; END_IF      END_IF
        IF bDev_MissingVoltage      THEN    DEV_Error.sErrorMessage := CONCAT(DEV_Error.sErrorMessage, 'Missing Voltage; ');            IF DEV_Error.ErrorPriority > 10  OR DEV_Error.ErrorPriority = 0 THEN DEV_Error.ErrorPriority := 10; END_IF      END_IF
        DEV_Error.bError := TRUE;
    ELSE
        DEV_Error.bError := FALSE;
        DEV_Error.sErrorMessage := '';
    END_IF

END_IF

//FB Instances
EL2819_Error(
    En                  := TRUE,
    iTerminal_ID        := iTerminal_ID,
    bWcState            := WcState_WcState,
    uiInfoData_State    := InfoData_State,
    pErrorSystem        := ErrorSystem,
    bError              => bError,
);

CH1_Error (
    En                  :=  En,
    bError              :=  ,
    sErrorMessage       :=  ,
    ErrorPriority       :=  ,
    iTerminal_ID        :=  iTerminal_ID,
    pErrorSystem        :=  ErrorSystem,
    EnO                 =>  ,
);

CH2_Error (
    En                  :=  En,
    bError              :=  ,
    sErrorMessage       :=  ,
    ErrorPriority       :=  ,
    iTerminal_ID        :=  iTerminal_ID,
    pErrorSystem        :=  ErrorSystem,
    EnO                 =>  ,
);

CH3_Error (
    En                  :=  En,
    bError              :=  ,
    sErrorMessage       :=  ,
    ErrorPriority       :=  ,
    iTerminal_ID        :=  iTerminal_ID,
    pErrorSystem        :=  ErrorSystem,
    EnO                 =>  ,
);

CH4_Error (
    En                  :=  En,
    bError              :=  ,
    sErrorMessage       :=  ,
    ErrorPriority       :=  ,
    iTerminal_ID        :=  iTerminal_ID,
    pErrorSystem        :=  ErrorSystem,
    EnO                 =>  ,
);

CH5_Error (
    En                  :=  En,
    bError              :=  ,
    sErrorMessage       :=  ,
    ErrorPriority       :=  ,
    iTerminal_ID        :=  iTerminal_ID,
    pErrorSystem        :=  ErrorSystem,
    EnO                 =>  ,
);

CH6_Error (
    En                  :=  En,
    bError              :=  ,
    sErrorMessage       :=  ,
    ErrorPriority       :=  ,
    iTerminal_ID        :=  iTerminal_ID,
    pErrorSystem        :=  ErrorSystem,
    EnO                 =>  ,
);

CH7_Error (
    En                  :=  En,
    bError              :=  ,
    sErrorMessage       :=  ,
    ErrorPriority       :=  ,
    iTerminal_ID        :=  iTerminal_ID,
    pErrorSystem        :=  ErrorSystem,
    EnO                 =>  ,
);

CH8_Error (
    En                  :=  En,
    bError              :=  ,
    sErrorMessage       :=  ,
    ErrorPriority       :=  ,
    iTerminal_ID        :=  iTerminal_ID,
    pErrorSystem        :=  ErrorSystem,
    EnO                 =>  ,
);

CH9_Error (
    En                  :=  En,
    bError              :=  ,
    sErrorMessage       :=  ,
    ErrorPriority       :=  ,
    iTerminal_ID        :=  iTerminal_ID,
    pErrorSystem        :=  ErrorSystem,
    EnO                 =>  ,
);

CH10_Error (
    En                  :=  En,
    bError              :=  ,
    sErrorMessage       :=  ,
    ErrorPriority       :=  ,
    iTerminal_ID        :=  iTerminal_ID,
    pErrorSystem        :=  ErrorSystem,
    EnO                 =>  ,
);

CH11_Error (
    En                  :=  En,
    bError              :=  ,
    sErrorMessage       :=  ,
    ErrorPriority       :=  ,
    iTerminal_ID        :=  iTerminal_ID,
    pErrorSystem        :=  ErrorSystem,
    EnO                 =>  ,
);

CH12_Error (
    En                  :=  En,
    bError              :=  ,
    sErrorMessage       :=  ,
    ErrorPriority       :=  ,
    iTerminal_ID        :=  iTerminal_ID,
    pErrorSystem        :=  ErrorSystem,
    EnO                 =>  ,
);

CH13_Error (
    En                  :=  En,
    bError              :=  ,
    sErrorMessage       :=  ,
    ErrorPriority       :=  ,
    iTerminal_ID        :=  iTerminal_ID,
    pErrorSystem        :=  ErrorSystem,
    EnO                 =>  ,
);

CH14_Error (
    En                  :=  En,
    bError              :=  ,
    sErrorMessage       :=  ,
    ErrorPriority       :=  ,
    iTerminal_ID        :=  iTerminal_ID,
    pErrorSystem        :=  ErrorSystem,
    EnO                 =>  ,
);

CH15_Error (
    En                  :=  En,
    bError              :=  ,
    sErrorMessage       :=  ,
    ErrorPriority       :=  ,
    iTerminal_ID        :=  iTerminal_ID,
    pErrorSystem        :=  ErrorSystem,
    EnO                 =>  ,
);

CH16_Error (
    En                  :=  En,
    bError              :=  ,
    sErrorMessage       :=  ,
    ErrorPriority       :=  ,
    iTerminal_ID        :=  iTerminal_ID,
    pErrorSystem        :=  ErrorSystem,
    EnO                 =>  ,
);

DEV_Error (
    En                  :=  En,
    bError              :=  ,
    sErrorMessage       :=  ,
    ErrorPriority       :=  ,
    iTerminal_ID        :=  iTerminal_ID,
    pErrorSystem        :=  ErrorSystem,
    EnO                 =>  ,
);

END_FUNCTION_BLOCK

// ---- tc_mca_std_lib/POUs/Hardware/EtherCAT_Terminals/Drives/EL2522.TcPOU
//EL2522 | 2-channel Puls/Dir terminal
FUNCTION_BLOCK EL2522

VAR_INPUT
    En: BOOL;
    iTerminal_ID : INT;
    ErrorSystem : POINTER TO ST_ErrorSystem;
END_VAR

VAR_OUTPUT
    EnO: BOOL;
    bError: BOOL;
END_VAR

VAR
    //WC_State is handled by NC, so NOT included here.
    InfoData_State AT %I*: UINT;

    //FB-s
    EL2522_Error    : FB_TerminalError;
END_VAR

(*
* TODO: Test on hardware
*)

EnO:=En;

EL2522_Error(
    En := TRUE,
    iTerminal_ID := iTerminal_ID,
    bWcState := FALSE,
    uiInfoData_State := InfoData_State,
    pErrorSystem := ErrorSystem,
    bError => bError,
);

END_FUNCTION_BLOCK

// ---- tc_mca_std_lib/POUs/Hardware/EtherCAT_Terminals/Drives/EL4134.TcPOU
//EL4134 | 4-channel analog output terminal, -10..+10V, 16 bit
FUNCTION_BLOCK EL4134

VAR_INPUT
    En: BOOL;
    iTerminal_ID : INT;
    ErrorSystem : POINTER TO ST_ErrorSystem;
END_VAR

VAR_OUTPUT
    EnO: BOOL;
    bError: BOOL;
END_VAR

VAR
    //WC_State is handled by NC, so NOT included here.
    InfoData_State AT %I*: UINT;

    //FB-s
    EL4134_Error    : FB_TerminalError;
END_VAR

(*
* TODO: Test on hardware
*)

EnO:=En;

EL4134_Error(
    En := TRUE,
    iTerminal_ID := iTerminal_ID,
    bWcState := FALSE,
    uiInfoData_State := InfoData_State,
    pErrorSystem := ErrorSystem,
    bError => bError,
);

END_FUNCTION_BLOCK

// ---- tc_mca_std_lib/POUs/Hardware/EtherCAT_Terminals/Drives/EL7037.TcPOU
//EL7037 | Stepper motor terminal, 24V DC, 1.5A
FUNCTION_BLOCK EL7037

VAR_INPUT
    En: BOOL;
    iTerminal_ID : INT;
    ErrorSystem : POINTER TO ST_ErrorSystem;
END_VAR

VAR_OUTPUT
    EnO: BOOL;
    bError: BOOL;
END_VAR

VAR
    //WC_State is handled by NC, so NOT included here.
    InfoData_State AT %I*: UINT;

    //FB-s
    EL7037_Error    : FB_TerminalError;
END_VAR

(*
* TODO: Test on hardware
*)

EnO:=En;

EL7037_Error(
    En := TRUE,
    iTerminal_ID := iTerminal_ID,
    bWcState := FALSE,
    uiInfoData_State := InfoData_State,
    pErrorSystem := ErrorSystem,
    bError => bError,
);

END_FUNCTION_BLOCK

// ---- tc_mca_std_lib/POUs/Hardware/EtherCAT_Terminals/Drives/EL7041_0052.TcPOU
//EL7041-0052 | Stepper motor terminal, 50V DC, 5A
FUNCTION_BLOCK EL7041_0052

VAR_INPUT
    En: BOOL;
    iTerminal_ID : INT;
    ErrorSystem : POINTER TO ST_ErrorSystem;
END_VAR

VAR_OUTPUT
    EnO: BOOL;
    bError: BOOL;
END_VAR

VAR
    //WC_State is handled by NC, so NOT included here.
    InfoData_State AT %I*: UINT;

    //FB-s
    EL7041_Error    : FB_TerminalError;
END_VAR

(*
* TODO: Test on hardware
*)

EnO:=En;

EL7041_Error(
    En := TRUE,
    iTerminal_ID := iTerminal_ID,
    bWcState := FALSE,
    uiInfoData_State := InfoData_State,
    pErrorSystem := ErrorSystem,
    bError => bError,
);

END_FUNCTION_BLOCK

// ---- tc_mca_std_lib/POUs/Hardware/EtherCAT_Terminals/Drives/EL7047.TcPOU
//EL7037 | Stepper motor terminal, 50V DC, 5A, Vector Control, Incremental Encoder
FUNCTION_BLOCK EL7047

VAR_INPUT
    En: BOOL;
    iTerminal_ID : INT;
    ErrorSystem : POINTER TO ST_ErrorSystem;
END_VAR

VAR_OUTPUT
    EnO: BOOL;
    bError: BOOL;
END_VAR

VAR
    //WC_State is handled by NC, so NOT included here.
    InfoData_State AT %I*: UINT;

    //FB-s
    EL7047_Error    : FB_TerminalError;
END_VAR

EnO:=En;

EL7047_Error(
    En := TRUE,
    iTerminal_ID := iTerminal_ID,
    bWcState := FALSE,
    uiInfoData_State := InfoData_State,
    pErrorSystem := ErrorSystem,
    bError => bError,
);

END_FUNCTION_BLOCK

// ---- tc_mca_std_lib/POUs/Hardware/EtherCAT_Terminals/Drives/EL7211.TcPOU
//EL7211 | Servo terminal, for resolver, 50V DC, 4.5Arms
FUNCTION_BLOCK EL7211

VAR_INPUT
    En: BOOL;
    iTerminal_ID : INT;
    ErrorSystem : POINTER TO ST_ErrorSystem;
END_VAR

VAR_OUTPUT
    EnO: BOOL;
    bError: BOOL;
END_VAR

VAR
    //WC_State is handled by NC, so NOT included here.
    InfoData_State AT %I*: UINT;

    //FB-s
    EL7211_Error    : FB_TerminalError;
END_VAR

(*
* TODO: Test on hardware
*)

EnO:=En;

EL7211_Error(
    En := TRUE,
    iTerminal_ID := iTerminal_ID,
    bWcState := FALSE,
    uiInfoData_State := InfoData_State,
    pErrorSystem := ErrorSystem,
    bError => bError,
);

END_FUNCTION_BLOCK

// ---- tc_mca_std_lib/POUs/Hardware/EtherCAT_Terminals/Feedback_Terminals/EL5002.TcPOU
//EL5002 | 2-chennel SSI absolute encoder terminal
FUNCTION_BLOCK EL5002

VAR_INPUT
    En: BOOL;
    iTerminal_ID : INT;
    ErrorSystem : POINTER TO ST_ErrorSystem;
END_VAR

VAR_OUTPUT
    EnO: BOOL;
    bError: BOOL;
END_VAR

VAR
    //WC_State is handled by NC, so NOT included here.
    InfoData_State AT %I*: UINT;

    //FB-s
    EL5002_Error    : FB_TerminalError;
END_VAR

(*
* TODO: Test on hardware
*)

EnO:=En;

EL5002_Error(
    En := TRUE,
    iTerminal_ID := iTerminal_ID,
    bWcState := FALSE,
    uiInfoData_State := InfoData_State,
    pErrorSystem := ErrorSystem,
    bError => bError,
);

END_FUNCTION_BLOCK

// ---- tc_mca_std_lib/POUs/Hardware/EtherCAT_Terminals/Feedback_Terminals/EL5021.TcPOU
//EL5021 | 1-channel Sin/Cos encoder
FUNCTION_BLOCK EL5021

VAR_INPUT
    En              : BOOL;
    iTerminal_ID    : INT;
    ErrorSystem     : POINTER TO ST_ErrorSystem;
END_VAR

VAR_OUTPUT
    EnO     : BOOL;
    bError  : BOOL;
END_VAR

VAR
    //WC_State is handled by NC, so NOT included here.
    InfoData_State      AT %I*  : UINT;

    //FB-s
    EL5021_Error    : FB_TerminalError;
END_VAR

(*
* TODO: Test on hardware
*)
EnO:=En;

//Error FB instances
EL5021_Error(
    En                  := TRUE,
    iTerminal_ID        := iTerminal_ID,
    bWcState            := FALSE,
    uiInfoData_State    := InfoData_State,
    pErrorSystem        := ErrorSystem,
    bError => bError,
);

END_FUNCTION_BLOCK

// ---- tc_mca_std_lib/POUs/Hardware/EtherCAT_Terminals/Feedback_Terminals/EL5042.TcPOU
//EL5042 | 2-channel BiSS-C absolute encoder terminal
FUNCTION_BLOCK EL5042

VAR_INPUT
    En: BOOL;
    iTerminal_ID    : INT;
    ErrorSystem     : POINTER TO ST_ErrorSystem;
END_VAR

VAR_OUTPUT
    EnO     : BOOL;
    bError  : BOOL;
END_VAR

VAR
    //WC_State is handled by NC, so NOT included here.
    InfoData_State      AT %I*  : UINT;

    //FB-s
    EL5042_Error    : FB_TerminalError;
END_VAR

(*
* TODO: Test on hardware
*)
EnO:=En;

//Error FB instances
EL5042_Error(
    En := TRUE,
    iTerminal_ID := iTerminal_ID,
    bWcState := FALSE,
    uiInfoData_State := InfoData_State,
    pErrorSystem := ErrorSystem,
    bError => bError,
);

END_FUNCTION_BLOCK

// ---- tc_mca_std_lib/POUs/Hardware/EtherCAT_Terminals/Feedback_Terminals/EL5101.TcPOU
// EL5101 | 1-channel incremental encoder terminal, 5V, RS422
FUNCTION_BLOCK EL5101

VAR_INPUT
    En              : BOOL;
    iTerminal_ID    : INT;
    ErrorSystem     : POINTER TO ST_ErrorSystem;
END_VAR

VAR_OUTPUT
    EnO     : BOOL;
    bError  : BOOL;
END_VAR

VAR
    //WC_State is handled by NC, so NOT included here.
    InfoData_State      AT %I* : UINT;

    //FB-s
    EL5101_Error    : FB_TerminalError;
END_VAR

(*
* TODO: Channel Status word (Connected to NC -> Not needed )
*)
EnO:=En;

//Error FB instances
EL5101_Error(
    En                  := TRUE,
    iTerminal_ID        := iTerminal_ID,
    bWcState            := FALSE,
    uiInfoData_State    := InfoData_State,
    pErrorSystem        := ErrorSystem,
    bError              => bError,
);

END_FUNCTION_BLOCK

// ---- tc_mca_std_lib/POUs/Hardware/EtherCAT_Terminals/Feedback_Terminals/EL7201.TcPOU
//EL7201 | 1-chennel resolver terminal (ESS only use it for resolver input)
FUNCTION_BLOCK EL7201

VAR_INPUT
    En: BOOL;
    iTerminal_ID : INT;
    ErrorSystem : POINTER TO ST_ErrorSystem;
END_VAR

VAR_OUTPUT
    EnO: BOOL;
    bError: BOOL;
END_VAR

VAR
    //WC_State is handled by NC, so NOT included here.
    InfoData_State AT %I*: UINT;

    //FB-s
    EL7201_Error    : FB_TerminalError;
END_VAR

(*
* TODO: Test on hardware
*)

EnO:=En;

EL7201_Error(
    En := TRUE,
    iTerminal_ID := iTerminal_ID,
    bWcState := FALSE,
    uiInfoData_State := InfoData_State,
    pErrorSystem := ErrorSystem,
    bError => bError,
);

END_FUNCTION_BLOCK

// ---- tc_mca_std_lib/POUs/Hardware/EtherCAT_Terminals/System/EK1100.TcPOU
FUNCTION_BLOCK EK1100

VAR_INPUT
    En              : BOOL;
    iTerminal_ID    : INT;
    ErrorSystem     : POINTER TO ST_ErrorSystem;
END_VAR

VAR_OUTPUT
    EnO     : BOOL;
    bError  : BOOL;
END_VAR

VAR
    InfoData_State  AT %I*  : UINT;

    //FB-s
    EK1100_Error    : FB_TerminalError;
END_VAR

(*
* TODO: DONE!
*)
EnO:=En;

//Error FB instance
EK1100_Error(
    En                  := TRUE,
    iTerminal_ID        := iTerminal_ID,
    bWcState            := FALSE,
    uiInfoData_State    := InfoData_State,
    pErrorSystem        := ErrorSystem,
    bError              => bError,
);

END_FUNCTION_BLOCK

// ---- tc_mca_std_lib/POUs/Hardware/EtherCAT_Terminals/System/EK1110.TcPOU
FUNCTION_BLOCK EK1110

VAR_INPUT
    En              : BOOL;
    iTerminal_ID    : INT;
    ErrorSystem     : POINTER TO ST_ErrorSystem;
END_VAR

VAR_OUTPUT
    EnO     : BOOL;
    bError  : BOOL;
END_VAR

VAR
    InfoData_State  AT %I*  : UINT;

    //FB-s
    EK1110_Error    : FB_TerminalError;
END_VAR

(*
* TODO: DONE!
*)
EnO:=En;

//Error FB instance
EK1110_Error(
    En                  := TRUE,
    iTerminal_ID        := iTerminal_ID,
    bWcState            := FALSE,
    uiInfoData_State    := InfoData_State,
    pErrorSystem        := ErrorSystem,
    bError              => bError,
);

END_FUNCTION_BLOCK

// ---- tc_mca_std_lib/POUs/Hardware/EtherCAT_Terminals/System/EL9410.TcPOU
//EL9410 | E-Bus power supplier and refresher, diagnostics
FUNCTION_BLOCK EL9410

VAR_INPUT
    En              : BOOL;
    iTerminal_ID    : INT;
    ErrorSystem     : POINTER TO ST_ErrorSystem;
END_VAR

VAR_OUTPUT
    EnO     : BOOL;
    bError  : BOOL;
END_VAR

VAR
    bUs_Undervoltage    AT %I*  : BOOL;
    bUp_Undervoltage    AT %I*  : BOOL;
    WcState_WcState     AT %I*  : BOOL;
    InfoData_State      AT %I*  : UINT;

    //FB-s
    EL9410_Error    : FB_TerminalError;
    PWR_Error       : FB_GenericError;
END_VAR

(*
* TODO: Status bits
*)
EnO:=En;

IF En THEN
    IF  bUs_Undervoltage OR bUp_Undervoltage THEN
        PWR_Error.sErrorMessage     := 'EL9410: ';
        IF bUs_Undervoltage     THEN    PWR_Error.sErrorMessage := CONCAT (PWR_Error.sErrorMessage, 'Us undervoltage; ');       IF PWR_Error.ErrorPriority > 5  OR PWR_Error.ErrorPriority = 0  THEN PWR_Error.ErrorPriority := 5;  END_IF  END_IF
        IF bUp_Undervoltage     THEN    PWR_Error.sErrorMessage := CONCAT (PWR_Error.sErrorMessage, 'Up undervoltage; ');       IF PWR_Error.ErrorPriority > 5  OR PWR_Error.ErrorPriority = 0  THEN PWR_Error.ErrorPriority := 5;  END_IF  END_IF
        PWR_Error.bError    := TRUE;
    ELSE
        PWR_Error.sErrorMessage := '';
        PWR_Error.bError        := FALSE;
    END_IF


END_IF

//Error FB instance
EL9410_Error(
    En                  := TRUE,
    iTerminal_ID        := iTerminal_ID,
    bWcState            := WcState_WcState,
    uiInfoData_State    := InfoData_State,
    pErrorSystem        := ErrorSystem,
    bError              => bError,
);

PWR_Error (
    En                  := En,
    bError              := ,
    sErrorMessage       := ,
    ErrorPriority       := ,
    iTerminal_ID        := iTerminal_ID,
    pErrorSystem        := ErrorSystem,
    EnO                 => ,
);

END_FUNCTION_BLOCK

// ---- tc_mca_std_lib/POUs/Hardware/EtherCAT_Terminals/System/EL9505.TcPOU
//EL9505 | Power supply terminal 5V
FUNCTION_BLOCK EL9505

VAR_INPUT
    En              : BOOL;
    iTerminal_ID    : INT;
    ErrorSystem     : POINTER TO ST_ErrorSystem;
END_VAR

VAR_OUTPUT
    EnO     : BOOL;
    bError  : BOOL;
END_VAR

VAR
    bUoPwr_OK           AT %I*  : BOOL;
    bUo_Overload        AT %I*  : BOOL;
    WcState_WcState     AT %I*  : BOOL;
    InfoData_State      AT %I*  : UINT;

    //FB-s
    EL9505_Error    : FB_TerminalError;
    PWR_Error       : FB_GenericError;
END_VAR

(*
* TODO: Test on hardware
*)
EnO:=En;

IF En THEN
    IF  (NOT bUoPwr_OK) OR bUo_Overload THEN
        PWR_Error.sErrorMessage     := 'EL9505: ';
        IF NOT bUoPwr_OK    THEN    PWR_Error.sErrorMessage := CONCAT (PWR_Error.sErrorMessage, 'Output Voltage Error; ');      IF PWR_Error.ErrorPriority > 5  OR PWR_Error.ErrorPriority = 0  THEN PWR_Error.ErrorPriority := 5;  END_IF  END_IF
        IF bUo_Overload     THEN    PWR_Error.sErrorMessage := CONCAT (PWR_Error.sErrorMessage, 'Overload; ');                  IF PWR_Error.ErrorPriority > 5  OR PWR_Error.ErrorPriority = 0  THEN PWR_Error.ErrorPriority := 5;  END_IF  END_IF
        PWR_Error.bError    := TRUE;
    ELSE
        PWR_Error.sErrorMessage := '';
        PWR_Error.bError        := FALSE;
    END_IF

END_IF


//Error FB instance
EL9505_Error(
    En                  := TRUE,
    iTerminal_ID        := iTerminal_ID,
    bWcState            := WcState_WcState,
    uiInfoData_State    := InfoData_State,
    pErrorSystem        := ErrorSystem,
    bError              => bError,
);

PWR_Error (
    En                  := En,
    bError              := ,
    sErrorMessage       := ,
    ErrorPriority       := ,
    iTerminal_ID        := iTerminal_ID,
    pErrorSystem        := ErrorSystem,
    EnO                 => ,
);

END_FUNCTION_BLOCK

// ---- tc_mca_std_lib/POUs/Motion/Homing/FB_HomeDirect.TcPOU
FUNCTION_BLOCK FB_HomeDirect
VAR_INPUT
    En: BOOL;
    bReset: BOOL;
    bExecute: BOOL;
    fHomePosition:LREAL;
END_VAR
VAR_IN_OUT
    Axis: AXIS_REF;
END_VAR
VAR_OUTPUT
    EnO: BOOL;
    bBusy: BOOL;
    bDone: BOOL;
    bHomed:BOOL;
    bError: BOOL;
    nErrorId: UDINT;
END_VAR
VAR
    fbHome: MC_Home;
END_VAR

En:=EnO;
IF bReset THEN
    bError:=FALSE;
    nErrorId:=0;
END_IF

fbHome(
    Execute:=bExecute,
    Position:=fHomePosition,
    HomingMode:=MC_Direct,
    bCalibrationCam:=FALSE,
    Axis:=Axis
    );

bBusy:=fbHome.Busy;
bDone:=fbHome.Done;
bHomed:=Axis.Status.Homed;

bError:=fbHome.Error;

IF fbHome.Error THEN
  nErrorId:=fbHome.ErrorID;
END_IF

END_FUNCTION_BLOCK

// ---- tc_mca_std_lib/POUs/Motion/Homing/FB_HomeFinish.TcPOU
FUNCTION_BLOCK FB_HomeFinish
VAR_INPUT
    En: BOOL;
    bReset: BOOL;
    bExecute: BOOL;
    nCmdData: UINT;
    bSofLimEnableLow: BOOL:=TRUE;
    bSofLimEnableHigh: BOOL:=TRUE;
END_VAR
VAR_IN_OUT
    Axis: AXIS_REF;
END_VAR
VAR_OUTPUT
    EnO: BOOL;
    bBusy: BOOL;
    bDone: BOOL;
    bError: BOOL;
    nErrorId: UDINT;
END_VAR
VAR
    fbHomewriteSoftLimEnable:FB_HomeWriteSoftLimEnable;
    fbExecuteRiseEdge: R_TRIG;
    bExecuteWriteNC:BOOL:=FALSE;
    nState:INT:=0;
END_VAR

En:=EnO;
IF bReset THEN
    bError:=FALSE;
    nErrorId:=0;
END_IF

IF NOT bExecute THEN
  bExecuteWriteNC:=FALSE;
  fbHomewriteSoftLimEnable.bSofLimEnableLow:=bSofLimEnableLow;
  fbHomewriteSoftLimEnable.bSofLimEnableHigh:=bSofLimEnableHigh;
  nState:=0;
END_IF

fbExecuteRiseEdge(CLK:=bExecute);
IF fbExecuteRiseEdge.Q THEN
  bExecuteWriteNC:=TRUE;
  fbHomewriteSoftLimEnable.bSofLimEnableLow:=bSofLimEnableLow;
  fbHomewriteSoftLimEnable.bSofLimEnableHigh:=bSofLimEnableHigh;
END_IF

// Write to NC (disable soft limits)
fbHomewriteSoftLimEnable(
    En:=En,
    bExecute:=bExecuteWriteNC AND bExecute,
    Axis:=Axis,
    bReset:=bReset,
);

bBusy:=fbHomewriteSoftLimEnable.bBusy;
bDone:=fbHomewriteSoftLimEnable.bDone;

bError:=fbHomewriteSoftLimEnable.bError;
IF fbHomewriteSoftLimEnable.bError THEN
  nErrorId:=fbHomewriteSoftLimEnable.nErrorId;
END_IF

END_FUNCTION_BLOCK

// ---- tc_mca_std_lib/POUs/Motion/Homing/FB_HomeWriteSoftLimEnable.TcPOU
FUNCTION_BLOCK FB_HomeWriteSoftLimEnable
VAR_INPUT
    En: BOOL;
    bReset: BOOL;
    bExecute: BOOL;
    bSofLimEnableLow: BOOL:=TRUE;
    bSofLimEnableHigh: BOOL:=TRUE;
END_VAR
VAR_IN_OUT
    Axis: AXIS_REF;
END_VAR
VAR_OUTPUT
    EnO: BOOL;
    bBusy: BOOL;
    bDone: BOOL;
    bError: BOOL;
    nErrorId: UDINT;
END_VAR
VAR
    fbExecuteRiseEdge: R_TRIG;
    fbWriteSoftLimEnableLow:FB_WriteParameterInNc_v1_00;
    fbWriteSoftLimEnableHigh:FB_WriteParameterInNc_v1_00;
END_VAR

En:=EnO;
IF bReset THEN
    bError:=FALSE;
    nErrorId:=0;
END_IF

fbExecuteRiseEdge(CLK:=bExecute);

fbWriteSoftLimEnableLow(
    bExecute:=bExecute,
    nDeviceGroup:= 16#5000,
    nIndexOffset:= 16#B,
    nData:=BOOL_TO_DWORD(bSofLimEnableLow),
    Axis:= Axis);

fbWriteSoftLimEnableHigh(
    bExecute:=bExecute,
    nDeviceGroup:= 16#5000,
    nIndexOffset:= 16#C,
    nData:=BOOL_TO_DWORD(bSofLimEnableHigh),
    Axis:= Axis);

bBusy:=fbWriteSoftLimEnableLow.bBusy OR fbWriteSoftLimEnableHigh.bBusy;
bDone:=fbWriteSoftLimEnableLow.bDone AND fbWriteSoftLimEnableHigh.bDone AND bExecute;

bError:=fbWriteSoftLimEnableHigh.bError OR fbWriteSoftLimEnableLow.bError;
IF fbWriteSoftLimEnableHigh.bError THEN
  nErrorId:=fbWriteSoftLimEnableHigh.nErrorId;
ELSIF fbWriteSoftLimEnableLow.bError THEN
  nErrorId:=fbWriteSoftLimEnableLow.nErrorId;
END_IF

END_FUNCTION_BLOCK

// ---- tc_mca_std_lib/POUs/Motion/Homing/FB_HomePrepare.TcPOU
FUNCTION_BLOCK FB_HomePrepare
VAR_INPUT
    En: BOOL;
    bReset: BOOL;
    bExecute: BOOL;
    nCmdData: UINT;
END_VAR
VAR_IN_OUT
    Axis: AXIS_REF;
END_VAR
VAR_OUTPUT
    EnO: BOOL;
    bBusy: BOOL;
    bDone: BOOL;
    bError: BOOL;
    nErrorId: UDINT;
    bSofLimEnableLowOriginal: BOOL:=TRUE;
    bSofLimEnableHighOriginal: BOOL:=TRUE;
    fVelocityToCam: LREAL:=0;
    fVelocityFromCam: LREAL:=0;
END_VAR
VAR
    fbHomeReadSoftLimEnable:FB_HomeReadSoftLimEnable;
    fbHomeDisableSoftLimEnable:FB_HomeWriteSoftLimEnable;
    fbHomeReadNCVelocities: FB_HomeReadNcVelocities;
    fbHomeResetCalibrationFlag:MC_Home;   //Only used for reset of calibration flag
    fbExecuteRiseEdge: R_TRIG;
    bExecuteReadNC:BOOL:=FALSE;
    bExecuteWriteNC:BOOL:=FALSE;
    nState:INT:=0;
END_VAR

En:=EnO;
IF bReset THEN
    bError:=FALSE;
    nErrorId:=0;
END_IF

IF NOT bExecute THEN
  bExecuteReadNC:=FALSE;
  bExecuteWriteNC:=FALSE;
  nState:=0;
END_IF

fbExecuteRiseEdge(CLK:=bExecute);
IF fbExecuteRiseEdge.Q THEN
  bExecuteReadNC:=TRUE;
END_IF

// Read from NC
fbHomeReadNCVelocities(
  En:=En,
  bExecute:=bExecuteReadNC, // Actualy not needed for sequence 15 (set position only, no movement))
  bReset:=bReset,
  Axis:=Axis,
);

fbHomeReadSoftLimEnable(
    En:=En,
    bExecute:=bExecuteReadNC AND bExecute,
    Axis:=Axis,
    bReset:=bReset,
);

// Reset calibration flag
fbHomeResetCalibrationFlag(
  Execute:=bExecuteReadNC,
  HomingMode:=MC_ResetCalibration,
  Axis:=Axis
);

bSofLimEnableLowOriginal:=fbHomeReadSoftLimEnable.bSofLimEnableLow;
bSofLimEnableHighOriginal:=fbHomeReadSoftLimEnable.bSofLimEnableHigh;

fVelocityToCam:=fbHomeReadNCVelocities.fVelocityToCam;
fVelocityFromCam:=fbHomeReadNCVelocities.fVelocityFromCam;

IF bExecuteReadNC AND bExecute AND fbHomeReadSoftLimEnable.bDone THEN
    fbHomeDisableSoftLimEnable.bSofLimEnableHigh:=FALSE;
    fbHomeDisableSoftLimEnable.bSofLimEnableLow:=FALSE;
    bExecuteWriteNC:=TRUE; //Always write (only needed if enabled actually)
END_IF

// Write to NC (disable soft limits)
fbHomeDisableSoftLimEnable(
    En:=En,
    bExecute:=bExecuteWriteNC AND bExecute,
    Axis:=Axis,
    bReset:=bReset,
);

bBusy:=fbHomeReadSoftLimEnable.bBusy OR fbHomeDisableSoftLimEnable.bBusy OR fbHomeReadNCVelocities.bBusy OR fbHomeResetCalibrationFlag.Busy;
bDone:=fbHomeReadSoftLimEnable.bDone AND fbHomeDisableSoftLimEnable.bDone AND fbHomeReadNCVelocities.bDone AND fbHomeResetCalibrationFlag.Done AND bExecute;

bError:=fbHomeReadSoftLimEnable.bError OR fbHomeDisableSoftLimEnable.bError OR fbHomeReadNCVelocities.bError OR fbHomeResetCalibrationFlag.Error;
IF fbHomeReadSoftLimEnable.bError THEN
  nErrorId:=fbHomeReadSoftLimEnable.nErrorId;
ELSIF fbHomeDisableSoftLimEnable.bError THEN
  nErrorId:=fbHomeDisableSoftLimEnable.nErrorId;
ELSIF fbHomeResetCalibrationFlag.Error THEN
  nErrorId:=fbHomeResetCalibrationFlag.ErrorId;
END_IF

END_FUNCTION_BLOCK

// ---- tc_mca_std_lib/POUs/Motion/Homing/FB_HomeReadSoftLimEnable.TcPOU
FUNCTION_BLOCK FB_HomeReadSoftLimEnable
VAR_INPUT
    En: BOOL;
    bReset: BOOL;
    bExecute: BOOL;
END_VAR
VAR_IN_OUT
    Axis: AXIS_REF;
END_VAR
VAR_OUTPUT
    EnO: BOOL;
    bBusy: BOOL;
    bDone: BOOL;
    bError: BOOL;
    nErrorId: UDINT;
    bSofLimEnableLow: BOOL:=TRUE;
    bSofLimEnableHigh: BOOL:=TRUE;
END_VAR
VAR
    fbReadSoftLimEnableLow:FB_ReadParameterInNc_v1_00;
    fbReadSoftLimEnableHigh:FB_ReadParameterInNc_v1_00;
END_VAR

En:=EnO;
IF bReset THEN
    bError:=FALSE;
    nErrorId:=0;
END_IF

fbReadSoftLimEnableLow(
    bExecute:=bExecute,
    nDeviceGroup:= 16#5000,
    nIndexOffset:= 16#B,
    Axis:= Axis);

fbReadSoftLimEnableHigh(
    bExecute:=bExecute,
    nDeviceGroup:= 16#5000,
    nIndexOffset:= 16#C,
    Axis:= Axis);

bSofLimEnableLow:=DWORD_TO_BOOL(fbReadSoftLimEnableLow.nData);
bSofLimEnableHigh:=DWORD_TO_BOOL(fbReadSoftLimEnableHigh.nData);

bBusy:=fbReadSoftLimEnableLow.bBusy OR fbReadSoftLimEnableHigh.bBusy;
bDone:=fbReadSoftLimEnableLow.bDone AND fbReadSoftLimEnableHigh.bDone AND bExecute;

bError:=fbReadSoftLimEnableLow.bError OR fbReadSoftLimEnableHigh.bError;
IF fbReadSoftLimEnableLow.bError THEN
  nErrorId:=fbReadSoftLimEnableLow.nErrorId;
ELSIF fbReadSoftLimEnableHigh.bError THEN
  nErrorId:=fbReadSoftLimEnableHigh.nErrorId;
END_IF

END_FUNCTION_BLOCK

// ---- tc_mca_std_lib/POUs/Motion/Homing/FB_HomeToSwitch.TcPOU
FUNCTION_BLOCK FB_HomeToSwitch
VAR_INPUT
    En: BOOL;
    bReset: BOOL;
    bExecute: BOOL;
    bCamSensor:BOOL;
    nSearchDirTwoardsCam: MC_Direction;
    nSearchDirOffCam: MC_Direction;
    fHomePosition:LREAL;
    fVelocityToCamNC: LREAL; //Velcoity when searching for cam
    fVelocityFromCamNC: LREAL; // Velocity after found cam (searching for next signal transition)
END_VAR
VAR_IN_OUT
    Axis: AXIS_REF;
END_VAR
VAR_OUTPUT
    EnO: BOOL;
    bBusy: BOOL;
    bDone: BOOL;
    bHomed:BOOL;
    bError: BOOL;
    nErrorId: UDINT;
END_VAR
VAR
    fbHome: MC_Home;
    fbWriteHomeDirCamToNC:FB_WriteParameterInNc_v1_00;
    fbWriteHomeDirSyncToNC:FB_WriteParameterInNc_v1_00;
    fbWriteHomeModeToNC:FB_WriteParameterInNc_v1_00;
    fbWriteHomeVelocitiesToNC: FB_HomeWriteNcVelocities;
    bConfigNCDone:BOOL:=FALSE;
    fbRTrigg: R_TRIG;
END_VAR

En:=EnO;
IF bReset THEN
    bConfigNCDone:=FALSE;
    bError:=FALSE;
    nErrorId:=0;
END_IF

//Start preparation of NC if rising edge on bExecute
fbRTrigg(CLK:=bExecute);
IF fbRTrigg.Q THEN
    bConfigNCDone:=FALSE;
END_IF


fbWriteHomeDirCamToNC(
    bExecute:=bExecute AND NOT bConfigNCDone,
    nDeviceGroup:=16#5000,
    nIndexOffset:=16#101,   //Direction for Calibration Cam Search
    nData:=BOOL_TO_DWORD(nSearchDirTwoardsCam=MC_Negative_Direction),//BOOL_TO_DWORD(NOT bSearchDirTwoardsCam),
    Axis:=Axis
);

fbWriteHomeDirSyncToNC(
    bExecute:= bExecute AND NOT bConfigNCDone,
    nDeviceGroup:=16#5000 ,
    nIndexOffset:=16#102 , //Direction for Sync Impuls Search
    nData:=BOOL_TO_DWORD(nSearchDirOffCam=MC_Negative_Direction),//BOOL_TO_DWORD(NOT bSearchDirOffCam),
    Axis:= Axis
);

fbWriteHomeModeToNC(
    bExecute:=bExecute AND NOT bConfigNCDone,
    nDeviceGroup:=16#5000,
    nIndexOffset:=16#107,  //Reference Mode
    nData:=1,
    Axis:=axis);

fbWriteHomeVelocitiesToNC(
  En:=En,
  bExecute:=bExecute AND NOT bConfigNCDone,
  bReset:=bReset,
  fVelocityFromCam:=fVelocityFromCamNC,
  fVelocityToCam:=fVelocityToCamNC,
  Axis:=Axis);

fbHome.bCalibrationCam:=bCamSensor;

fbHome(
    Execute:=bExecute AND bConfigNCDone(* AND NOT bError*),
    Position:=fHomePosition,
    HomingMode:=0,
    Axis:=Axis
    );
bBusy:=(fbHome.Busy OR (NOT bConfigNCDone AND bExecute));
bDone:=fbHome.Done AND bConfigNCDone;
bHomed:=Axis.Status.Homed;

IF (NOT bConfigNCDone) AND fbWriteHomeDirCamToNC.bDone AND fbWriteHomeDirSyncToNC.bDone AND fbWriteHomeModeToNC.bDone AND fbWriteHomeVelocitiesToNC.bDone THEN
  bConfigNCDone:=TRUE;
END_IF

//For some reason MC_HOME gives an Error for one cycle of NC-Task 1 SVB (10ms default..) so filter with bExecute
bError:=(fbHome.Error AND bExecute) OR fbWriteHomeDirCamToNC.bError OR fbWriteHomeDirSyncToNC.bError OR fbWriteHomeModeToNC.bError OR fbWriteHomeVelocitiesToNC.bError;

IF (fbHome.Error AND bExecute) THEN
  nErrorId:=fbHome.ErrorID;
ELSIF fbWriteHomeDirCamToNC.bError THEN
  nErrorId:=fbWriteHomeDirCamToNC.nErrorId;
ELSIF fbWriteHomeDirSyncToNC.bError THEN
  nErrorId:=fbWriteHomeDirSyncToNC.nErrorId;
ELSIF fbWriteHomeModeToNC.bError THEN
  nErrorId:=fbWriteHomeModeToNC.nErrorId;
ELSIF fbWriteHomeVelocitiesToNC.bError THEN
  nErrorId:=fbWriteHomeVelocitiesToNC.nErrorId;
END_IF

END_FUNCTION_BLOCK

// ---- tc_mca_std_lib/POUs/Motion/Homing/FB_HomeWriteNcVelocities.TcPOU
FUNCTION_BLOCK FB_HomeWriteNcVelocities
VAR_INPUT
    En: BOOL;
    bReset: BOOL;
    bExecute: BOOL;
    fVelocityToCam: LREAL;
    fVelocityFromCam: LREAL;
END_VAR
VAR_IN_OUT
    Axis: AXIS_REF;
END_VAR
VAR_OUTPUT
    EnO: BOOL;
    bBusy: BOOL;
    bDone: BOOL;
    bError: BOOL;
    nErrorId: UDINT;
END_VAR
VAR
    fbExecuteRiseEdge: R_TRIG;
    fbWriteVelocityToCam:FB_WriteFloatParameter;
    fbWriteVelocityFromCam:FB_WriteFloatParameter;
END_VAR

En:=EnO;
IF bReset THEN
    bError:=FALSE;
    nErrorId:=0;
END_IF

fbExecuteRiseEdge(CLK:=bExecute);

fbWriteVelocityToCam(
    bExecute:=bExecute,
    nDeviceGroup:= 16#4000,
    nIndexOffset:= 16#6,
    nData:=fVelocityToCam,
    Axis:= Axis);

fbWriteVelocityFromCam(
    bExecute:=bExecute,
    nDeviceGroup:= 16#4000,
    nIndexOffset:= 16#7,
    nData:=fVelocityFromCam,
    Axis:= Axis);

bBusy:=fbWriteVelocityFromCam.bBusy OR fbWriteVelocityToCam.bBusy;
bDone:=fbWriteVelocityFromCam.bDone AND fbWriteVelocityToCam.bDone AND bExecute;

bError:=fbWriteVelocityToCam.bError OR fbWriteVelocityFromCam.bError;
IF fbWriteVelocityToCam.bError THEN
  nErrorId:=fbWriteVelocityToCam.nErrorId;
ELSIF fbWriteVelocityFromCam.bError THEN
  nErrorId:=fbWriteVelocityFromCam.nErrorId;
END_IF

END_FUNCTION_BLOCK

// ---- tc_mca_std_lib/POUs/Motion/Homing/FB_HomeVirtual.TcPOU
FUNCTION_BLOCK FB_HomeVirtual
VAR_INPUT
    En: BOOL;
    bReset: BOOL;
    bExecute: BOOL;
    nCmdData: UINT;
    bLimitFwd: BOOL;
    bLimitBwd: BOOL;
    bHomeSensor: BOOL;
    fHomePosition:LREAL;
    nHomeRevOffset: UINT;
    nHomeProc: UINT;
END_VAR
VAR_IN_OUT
    Axis: AXIS_REF;
END_VAR
VAR_OUTPUT
    EnO: BOOL;
    bBusy: BOOL;
    bDone: BOOL;
    bHomed:BOOL;
    bError: BOOL;
    nErrorId: UDINT;
END_VAR
VAR
    fbHomeToSwitch: FB_HomeToSwitch;
    fbHomeDirect: FB_HomeDirect; //Only used for direct homing (set of position)
    fbMoveVelocity:MC_MoveVelocity;
    fbHomePrepare:FB_HomePrepare;
    fbHomeFinish:FB_HomeFinish;
    fbExecuteRiseEdge: R_TRIG;
    nHomingState:INT:=0;
    bExecuteHomeToSwitch:BOOL:=FALSE;
    bExecuteMoveVelocity:BOOL:=FALSE;
    bExecutePrepare: BOOL:=FALSE;
    bExecuteFinish: BOOL:=FALSE;
    bExecuteHomeDirect: BOOL;
    nHomeProcLocal: UINT;  //Ensure that nCmdData is not changed during sequence
    bSequenceReady:BOOL:=TRUE;
    bRestoreNCDataNeeded: BOOL:=FALSE;
END_VAR

EnO:=En;

IF bReset THEN
    bError:=FALSE;
    nErrorId:=0;
END_IF

// Reset when bExecute is low
IF NOT bExecute THEN
  nHomingState:=0;
  bSequenceReady:=TRUE;
  bExecuteHomeToSwitch:=FALSE;
  bExecuteHomeDirect:=FALSE;
  bExecuteMoveVelocity:=FALSE;
  bExecutePrepare:=FALSE;
  bExecuteFinish:=FALSE;
END_IF

//Reset at rinsing edge of bExecute
fbExecuteRiseEdge(CLK:=bExecute);
IF fbExecuteRiseEdge.Q THEN
  nHomeProcLocal:=nHomeProc; //Ensure that nHomeProc is not changed during sequence (nCmdData will only be read at a rising edge of bExecute)
  bSequenceReady:=FALSE;
  bExecutePrepare:=TRUE;
  bRestoreNCDataNeeded:=FALSE;
  //Check if valid nCmdDataLocal
  CASE nHomeProcLocal OF
    1:
    2:
    3:
    4:
    15:
    ELSE //nCmdData not valid
      bError:=TRUE;
      nErrorId:=16#4FFF;
  END_CASE
END_IF

//############# Prepare for homing (Read from NC and reset homed flag)
fbHomePrepare(
  En:=En,
  bExecute:=bExecutePrepare AND NOT bError, // Not needed for sequence 15 (set position only, no movement))
  bReset:=bReset,
  Axis:=Axis,
);

//############# Homing Sequences:
CASE nCmdDataLocal OF

   1: // Home to low limit switch
       CASE nHomingState OF
          0:
            bHomed:=Axis.Status.Homed;
            // Wait for read of velocities from NC and reset of calibration flag
            IF fbHomePrepare.bDone AND bExecute AND NOT bSequenceReady THEN
              bRestoreNCDataNeeded:=TRUE;
              IF bLimitBwd THEN
                nHomingState:=1;
              ELSE
                nHomingState:=2;  //Standing on limit switch go direct to state 2
              END_IF
            END_IF
          1: // wait for reach low limit then trigger fbHomeToSwitch
            bHomed:=FALSE;
            bSequenceReady:=FALSE;
            fbMoveVelocity.Velocity:=ABS(fbHomePrepare.fVelocityToCam);
            fbMoveVelocity.Direction:=MC_Negative_Direction;
            bExecuteMoveVelocity:=bExecute;  // Execute MC_MoveVelocity
            IF NOT bLimitBwd AND NOT fbMoveVelocity.Busy AND Axis.Status.NotMoving THEN //MC_MoveVelocity.Busy goes down when ramp down initiates (not ends).
              nHomingState:=2;
            END_IF
          2: // Wait for fbHomeToSwitch
            bHomed:=FALSE;
            bSequenceReady:=FALSE;
            bExecuteMoveVelocity:=FALSE;
            bExecuteHomeToSwitch:=TRUE;
            fbHomeToSwitch.nSearchDirTwoardsCam:=MC_Positive_Direction;
            fbHomeToSwitch.nSearchDirOffCam:=MC_Positive_Direction;
            fbHomeToSwitch.fVelocityToCamNC:=fbHomePrepare.fVelocityToCam; // High speed
            fbHomeToSwitch.fVelocityFromCamNC:=fbHomePrepare.fVelocityFromCam;  // Low speed
            fbHomeToSwitch.bCamSensor:=NOT bLimitBwd;
            IF fbHomeToSwitch.bDone THEN
              nHomingState:=3;
              bExecuteFinish:=TRUE;
              fbHomeFinish.bSofLimEnableHigh:=fbHomePrepare.bSofLimEnableHighOriginal;
              fbHomeFinish.bSofLimEnableLow:=fbHomePrepare.bSofLimEnableLowOriginal;
            END_IF;
          3: // restore softlimit enable
            bHomed:=FALSE;
            bSequenceReady:=FALSE;
            IF fbHomeFinish.bDone THEN
              bRestoreNCDataNeeded:=FALSE;
              bSequenceReady:=TRUE;
              nHomingState:=0;
              bHomed:=Axis.Status.Homed;
            END_IF;
       END_CASE;

   2: // Home to high limit switch
       CASE nHomingState OF
          0:
            bHomed:=Axis.Status.Homed;
            // Wait for read of velocities from NC and reset of calibration flag
            IF fbHomePrepare.bDone AND bExecute AND NOT bSequenceReady THEN
              bRestoreNCDataNeeded:=TRUE;
              IF bLimitFwd THEN
                nHomingState:=1;
              ELSE
                nHomingState:=2;  //Standing on limit switch go direct to state 2
              END_IF
            END_IF
          1: // wait for reach low limit then trigger fbHomeToSwitch
            bHomed:=FALSE;
            bSequenceReady:=FALSE;
            fbMoveVelocity.Velocity:=ABS(fbHomePrepare.fVelocityToCam);
            fbMoveVelocity.Direction:=MC_Positive_Direction;
            bExecuteMoveVelocity:=bExecute;  // Execute MC_MoveVelocity
            IF NOT bLimitFwd AND NOT fbMoveVelocity.Busy AND Axis.Status.NotMoving THEN //MC_MoveVelocity.Busy goes down when ramp down initiates (not ends).
              nHomingState:=2;
            END_IF
          2: // Wait for fbHomeToSwitch
            bHomed:=FALSE;
            bSequenceReady:=FALSE;
            bExecuteMoveVelocity:=FALSE;
            bExecuteHomeToSwitch:=TRUE;
            fbHomeToSwitch.nSearchDirTwoardsCam:=MC_Negative_Direction;
            fbHomeToSwitch.nSearchDirOffCam:=MC_Negative_Direction;
            fbHomeToSwitch.fVelocityToCamNC:=fbHomePrepare.fVelocityToCam; // High speed
            fbHomeToSwitch.fVelocityFromCamNC:=fbHomePrepare.fVelocityFromCam;  // Low speed
            fbHomeToSwitch.bCamSensor:=NOT bLimitFwd;
            IF fbHomeToSwitch.bDone THEN
              nHomingState:=3;
              bExecuteFinish:=TRUE;
              fbHomeFinish.bSofLimEnableHigh:=fbHomePrepare.bSofLimEnableHighOriginal;
              fbHomeFinish.bSofLimEnableLow:=fbHomePrepare.bSofLimEnableLowOriginal;
            END_IF;
          3: // restore softlimit enable
            bHomed:=FALSE;
            bSequenceReady:=FALSE;
            IF fbHomeFinish.bDone THEN
              bRestoreNCDataNeeded:=FALSE;
              bSequenceReady:=TRUE;
              nHomingState:=0;
              bHomed:=Axis.Status.Homed;
            END_IF;
       END_CASE;

   3: // Home on bHomeSensor via bLimitBwd
       CASE nHomingState OF
          0:
            bHomed:=Axis.Status.Homed;
            // Wait for read of velocities from NC and reset of calibration flag
            IF fbHomePrepare.bDone AND bExecute AND NOT bSequenceReady THEN
              bRestoreNCDataNeeded:=TRUE;
              IF bLimitBwd THEN
                nHomingState:=1;
              ELSE
                nHomingState:=2;  //Standing on limit switch go direct to state 2
              END_IF
            END_IF
          1: // wait for reach low limit then trigger fbHomeToSwitch
            bHomed:=FALSE;
            bSequenceReady:=FALSE;
            fbMoveVelocity.Velocity:=ABS(fbHomePrepare.fVelocityToCam);
            fbMoveVelocity.Direction:=MC_Negative_Direction;
            bExecuteMoveVelocity:=bExecute;  // Execute MC_MoveVelocity
            IF NOT bLimitBwd AND NOT fbMoveVelocity.Busy AND Axis.Status.NotMoving THEN //MC_MoveVelocity.Busy goes down when ramp down initiates (not ends).
              nHomingState:=2;
            END_IF
          2: // Wait for fbHomeToSwitch
            bHomed:=FALSE;
            bSequenceReady:=FALSE;
            bExecuteMoveVelocity:=FALSE;
            bExecuteHomeToSwitch:=TRUE;
            fbHomeToSwitch.nSearchDirTwoardsCam:=MC_Positive_Direction;
            fbHomeToSwitch.nSearchDirOffCam:=MC_Positive_Direction;
            fbHomeToSwitch.fVelocityToCamNC:=fbHomePrepare.fVelocityToCam; // High speed
            fbHomeToSwitch.fVelocityFromCamNC:=fbHomePrepare.fVelocityFromCam;  // Low speed
            fbHomeToSwitch.bCamSensor:=bHomeSensor;
            IF fbHomeToSwitch.bDone THEN
              nHomingState:=3;
              bExecuteFinish:=TRUE;
              fbHomeFinish.bSofLimEnableHigh:=fbHomePrepare.bSofLimEnableHighOriginal;
              fbHomeFinish.bSofLimEnableLow:=fbHomePrepare.bSofLimEnableLowOriginal;
            END_IF;
          3: // restore softlimit enable
            bHomed:=FALSE;
            bSequenceReady:=FALSE;
            IF fbHomeFinish.bDone THEN
              bRestoreNCDataNeeded:=FALSE;
              bSequenceReady:=TRUE;
              nHomingState:=0;
              bHomed:=Axis.Status.Homed;
            END_IF;
       END_CASE;
    4:  // Home on bHomeSensor via bLimitFwd
       CASE nHomingState OF
          0:
            bHomed:=Axis.Status.Homed;
            // Wait for read of velocities from NC and reset of calibration flag
            IF fbHomePrepare.bDone AND bExecute AND NOT bSequenceReady THEN
              bRestoreNCDataNeeded:=TRUE;
              IF bLimitFwd THEN
                nHomingState:=1;
              ELSE
                nHomingState:=2;  //Standing on limit switch go direct to state 2
              END_IF
            END_IF
          1: // wait for reach low limit then trigger fbHomeToSwitch
            bHomed:=FALSE;
            bSequenceReady:=FALSE;
            fbMoveVelocity.Velocity:=ABS(fbHomePrepare.fVelocityToCam);
            fbMoveVelocity.Direction:=MC_Positive_Direction;
            bExecuteMoveVelocity:=bExecute;  // Execute MC_MoveVelocity
            IF NOT bLimitFwd AND NOT fbMoveVelocity.Busy AND Axis.Status.NotMoving THEN //MC_MoveVelocity.Busy goes down when ramp down initiates (not ends).
              nHomingState:=2;
            END_IF
          2: // Wait for fbHomeToSwitch
            bHomed:=FALSE;
            bSequenceReady:=FALSE;
            bExecuteMoveVelocity:=FALSE;
            bExecuteHomeToSwitch:=TRUE;
            fbHomeToSwitch.nSearchDirTwoardsCam:=MC_Negative_Direction;
            fbHomeToSwitch.nSearchDirOffCam:=MC_Negative_Direction;
            fbHomeToSwitch.fVelocityToCamNC:=fbHomePrepare.fVelocityToCam; // High speed
            fbHomeToSwitch.fVelocityFromCamNC:=fbHomePrepare.fVelocityFromCam;  // Low speed
            fbHomeToSwitch.bCamSensor:=bHomeSensor;
            IF fbHomeToSwitch.bDone THEN
              nHomingState:=3;
              bExecuteFinish:=TRUE;
              fbHomeFinish.bSofLimEnableHigh:=fbHomePrepare.bSofLimEnableHighOriginal;
              fbHomeFinish.bSofLimEnableLow:=fbHomePrepare.bSofLimEnableLowOriginal;
            END_IF;
          3: // Restore softlimit enable
            bHomed:=FALSE;
            bSequenceReady:=FALSE;
            IF fbHomeFinish.bDone THEN
              bRestoreNCDataNeeded:=FALSE;
              bSequenceReady:=TRUE;
              nHomingState:=0;
              bHomed:=Axis.Status.Homed;
            END_IF;
       END_CASE;

   15: //Set current position (simplest homing sequence)
     bExecuteHomeDirect:=bExecute;
     bHomed:=Axis.Status.Homed;
     IF fbHomeDirect.bDone THEN  //Homing ready
       bExecuteHomeDirect:=FALSE;
       bSequenceReady:=TRUE;
     END_IF

ELSE
  fbHomeToSwitch.bCamSensor:=FALSE;
  bHomed:=Axis.Status.Homed;
END_CASE;

// Main homing block
fbHomeToSwitch(
    bExecute:=bExecuteHomeToSwitch AND bExecute AND NOT bError AND NOT bExecuteHomeDirect AND NOT bExecuteMoveVelocity,
    bReset:=bReset,
    fHomePosition:=fHomePosition,
    Axis:=Axis
);

// Approach limit switch (error if MC_Home is used)
fbMoveVelocity(
    Execute:= bExecuteMoveVelocity AND bExecute AND NOT bError AND NOT bExecuteHomeToSwitch AND NOT bExecuteHomeDirect,
    Axis:=Axis
);

// No sequence, just set position value (nCmdDataLocal=15). Can not run if fbHomeToSwitch is executed
fbHomeDirect(
    bExecute:=bExecuteHomeDirect AND bExecute AND NOT bError  AND NOT bExecuteHomeToSwitch AND NOT bExecuteMoveVelocity,
    bReset:=bReset,
    fHomePosition:=fHomePosition,
    Axis:=Axis
);


//############# Finish homing

IF NOT bexecute AND bRestoreNCDataNeeded THEN  //If homing is aborted restore is needed
    bExecuteFinish:=TRUE;
    IF fbHomeFinish.bDone THEN
      bExecuteFinish:=FALSE;
      bRestoreNCDataNeeded:=FALSE;
    END_IF
END_IF

fbHomeFinish(
  En:=En,
  bExecute:=bExecuteFinish,
  bReset:=bReset,
  Axis:=Axis,
);

// Error handling
IF NOT bError THEN
  IF fbHomeToSwitch.bError THEN
    bError:=fbHomeToSwitch.bError;
    nErrorId:=fbHomeToSwitch.nErrorId;
  ELSIF fbHomeDirect.bError THEN
    bError:=fbHomeDirect.bError;
    nErrorId:=fbHomeDirect.nErrorId;
  ELSIF fbMoveVelocity.Error THEN
    bError:=fbMoveVelocity.Error;
    nErrorId:=fbMoveVelocity.ErrorId;
  END_IF;
END_IF

// Done and busy bit
bDone:=bSequenceReady AND bExecute;
bBusy:=NOT bSequenceReady;

RETURN;

END_FUNCTION_BLOCK

// ---- GlobalTextList.TcGTLO
TEXTLIST GlobalTextList
  951 = '%2.2f'
  878 = '%d'
  706 = '%i'
  940 = '%x'
  703 = 'Acknowledge'
  710 = 'Active:'
  952 = 'actPos'
  953 = 'actVel'
  110 = 'AXESMAX'
  107 = 'axisSel'
  945 = 'bBusy'
  950 = 'bBwEnabled'
  946 = 'bDone'
  943 = 'bEnabled'
  941 = 'bError'
  102 = 'bExecute'
  949 = 'bFwEnabled'
  297 = 'bGeared'
  948 = 'bHomed'
  947 = 'bResetDone'
  944 = 'bWarning'
  704 = 'Clear All'
  104 = 'ENABLE'
  106 = 'ENABLE BW'
  105 = 'ENABLE FW'
  109 = 'English'
  939 = 'errID'
  701 = 'Error #'
  705 = 'Error #:'
  702 = 'Error Log'
  707 = 'Errors:'
  955 = 'fAcceleration'
  956 = 'fDeceleration'
  957 = 'fPosition'
  708 = 'Free Entries:'
  954 = 'fVelocity'
  299 = 'gearIn'
  300 = 'gearOut'
  711 = 'Inactive:'
  116 = 'jogBw'
  117 = 'jogFw'
  298 = 'masterGear'
  111 = 'moveAbsolute'
  114 = 'moveModulo'
  113 = 'moveRelative'
  112 = 'moveVelocity'
  709 = 'Overflows:'
  942 = 'reset'
  115 = 'stop'
  108 = 'Test Language'
  103 = 'toggle'
END_TEXTLIST

// ---- tc_mca_std_lib/POUs/VISUs/Error_Log_Visu.TcVIS
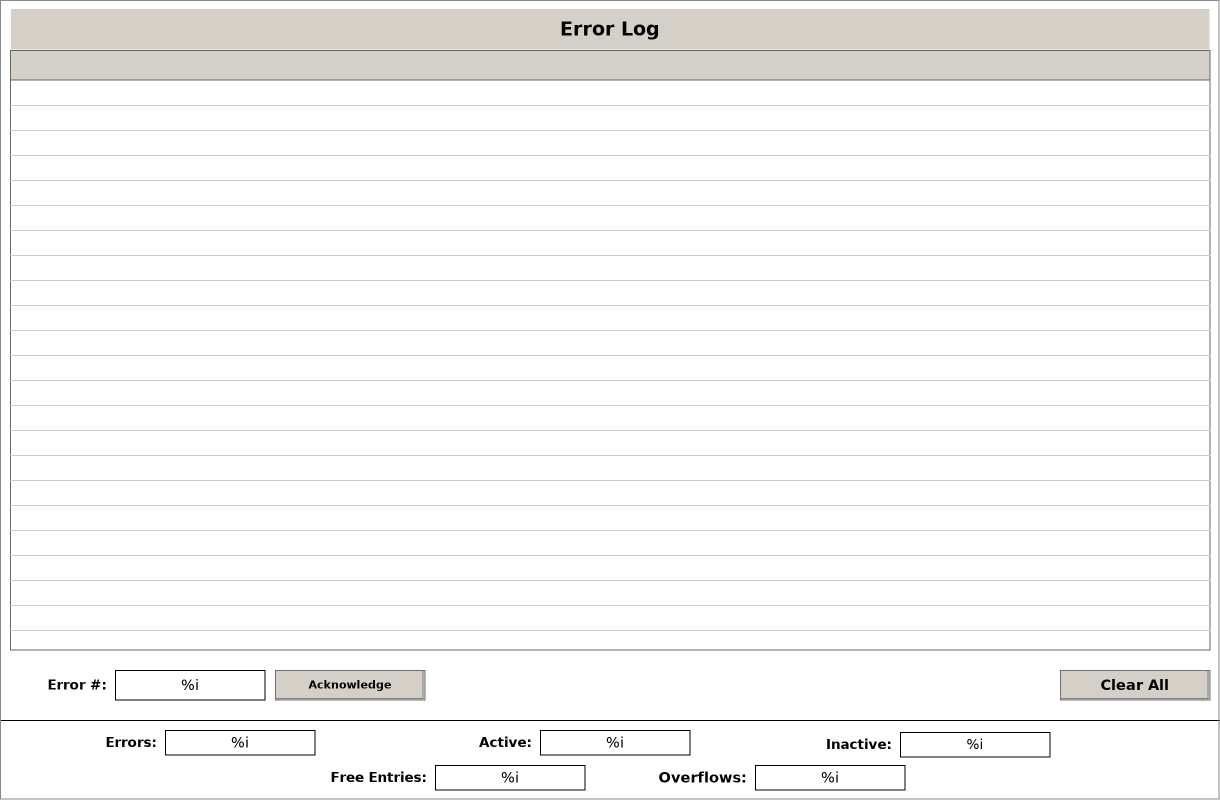
VISUALIZATION Error_Log_Visu  // 1220x800
    Table (10,50 1200x600), data array: MAIN.fbErrorSystem.ErrorSystem.aErrorData
        p1128707560: cSizeOfErrorData
        p1137915858: MAIN.fbErrorSystem.nTableRowIndex
        p1822360349: MAIN.fbErrorSystem.bValidSelection
        p3854506369: MAIN.fbErrorSystem.ErrorSystem.aErrorData[INDEX].ErrorNum
        p1892666644: MAIN.fbErrorSystem.ErrorSystem.aErrorData[INDEX].ErrorState
        p338671338: MAIN.fbErrorSystem.ErrorSystem.aErrorData[INDEX].iTerminalID
        p2170511999: MAIN.fbErrorSystem.ErrorSystem.aErrorData[INDEX].sDateTimeOn
        p3723444502: MAIN.fbErrorSystem.ErrorSystem.aErrorData[INDEX].sDateTimeOff
        p1218418051: MAIN.fbErrorSystem.ErrorSystem.aErrorData[INDEX].sErrorMessage
        p746581629: MAIN.fbErrorSystem.ErrorSystem.aErrorData[INDEX].ErrorPriority
        p2232123230: Error #
        p1755163831: Terminal ID
        p4092479075: Encountered on:
        p2237128397: Disapeared on:
        p505689113: Description
    Rectangle (11,9 1198x40), "Error Log"
    Button (275,670 150x30), "Acknowledge"
        tap MAIN.fbErrorSystem.bACK
        OnMouseUp: execute { MAIN.fbErrorSystem.nErrorNum := 0; }
    Button (1060,670 150x30), "Clear All"
        tap MAIN.fbErrorSystem.bReset
    Label (10,670 100x30), "Error #:"
    RoundedRectangle (115,670 150x30), "%i", text variable: MAIN.fbErrorSystem.nSelectedError
        OnMouseUp: write MAIN.fbErrorSystem.nErrorNum via Default, min 0
    Line (0,720) (1220,720)
    Label (10,730 150x25), "Errors:"
    Label (280,765 150x25), "Free Entries:"
    Label (600,765 150x25), "Overflows:"
    RoundedRectangle (165,730 150x25), "%i", text variable: MAIN.fbErrorSystem.ErrorSystem.nNoError
    RoundedRectangle (435,765 150x25), "%i", text variable: MAIN.fbErrorSystem.nFreePos
    RoundedRectangle (755,765 150x25), "%i", text variable: MAIN.fbErrorSystem.ErrorSystem.nNoOverflow
    Label (385,730 150x25), "Active:"
    Label (745,732 150x25), "Inactive:"
    RoundedRectangle (540,730 150x25), "%i", text variable: MAIN.fbErrorSystem.ErrorSystem.nNoActive
    RoundedRectangle (900,732 150x25), "%i", text variable: MAIN.fbErrorSystem.ErrorSystem.nNoInactive
END_VISUALIZATION

// ---- tc_mca_std_lib/POUs/VISUs/languageSupport.TcTLO
TEXTLIST languageSupport
  axesAvailable = 'PLC Axes available: %d' | Test: 'Alt language'
  velocity = 'Velocity:'
  actposition = 'Actual Position:'
  enable = 'Enable Axis'
  enFW = 'Enable Forward'
  enBW = 'Enable Backward'
  axisSel = 'Axis Selected:'
  actVelocity = 'Actual Velocity:'
  errID = 'Error ID:'
  bEnabled = 'Axis Enabled'
  bWarning = 'Warning'
  bBusy = 'Busy'
  bDone = 'Command Done'
  bHomed = 'Calibrated'
  bFwEnabled = 'Fwd movement enabled'
  bBwEnabled = 'Bwd movement enabled'
  bError = 'Error'
  fVelocity = 'Target Velocity:' | Test: 'Geschwindigkeit:'
  fAcceleration = 'Target Accel.:'
  fDeceleration = 'Target Decel.:'
  fPosition = 'Target Position:'
  moveAbsolute = 'Absolute position move'
  toggle = 'Toggle'
  moveVelocity = 'Constant velocity move'
  bExecute = 'Motion function executed'
  moveRelative = 'Relative position move'
  moveModulo = 'Modulo position move'
  reset = 'Reset axis'
  stop = 'Stop motion'
  jogBw = 'Jog Backward'
  jogFw = 'Jog Forward'
  bGeared = 'In Gear'
  masterGear = 'Master Axis'
  gearRatio = 'Gear Ratio'
  gearIn = 'Gear In'
  gearOut = 'Gear Out'
  homeSensorNeg = 'Home to Sensor (Neg)'
  homeSensorPos = 'Home to Sensor (Pos)'
   = ''
END_TEXTLIST

